// TwinCAT 3 PLC project SFICrane
// ProgramVersion: 3.1.4023.0
// libraries:
//   Tc2_MC2, * (Beckhoff Automation GmbH)
//   Tc2_MC2_Drive, * (Beckhoff Automation GmbH)
//   Tc2_Standard, * (Beckhoff Automation GmbH)
//   Tc2_System, * (Beckhoff Automation GmbH)
//   Tc2_Utilities, * (Beckhoff Automation GmbH)
//   Tc3_Module, * (Beckhoff Automation GmbH)
// project tree:
//   AXIS CONTROL/ GVL_AXIS1.TcGVL, GVL_AXIS2.TcGVL (not stored), GVL_AXIS3.TcGVL, GVL_AXIS4.TcGVL, GVL_Safety_AXIS4.TcGVL, P_AxisControl.TcPOU, P_AxisControl_1.TcPOU, ST_MC_CMD.TcDUT (not stored), ST_MC_ParametersAxis.TcDUT (not stored), ST_MC_Status.TcDUT (not stored)
//   / GlobalTextList.TcGTLO, MAIN.TcPOU (not stored), PlcTask.TcTTO (not stored), Visualization Manager.TcVMO (not stored)
//   HMI/ HMI.TcVIS
//   INPUTS/Function Blocks/ FB_AnalogInputScaling.TcPOU (not stored), FB_JoystickInputScaling.TcPOU (not stored)
//   INPUTS/ G_Inputs.TcGVL, G_ScalingParameters.TcGVL (not stored), G_Sensors.TcGVL (not stored), P_Inputs.TcPOU
//   INPUTS/Struct/ ST_AnalogInput.TcDUT (not stored), ST_AnalogInputScaling.TcDUT (not stored), ST_AnalogInputStatus.TcDUT (not stored), ST_JoystickInputScaling.TcDUT (not stored), ST_Parameters.TcDUT (not stored)
//   MACHINE CONTROL/ G_MachineControl.TcGVL, P_MachineControl.TcPOU (unreadable)
//   MACHINE CONTROL/KinematicFunctions2d/ cosd.TcPOU (not stored), FB_Forward.TcPOU, GVL_InverseKinematics.TcGVL, FB_Inverse.TcPOU (not stored), rt_ceild.TcPOU (not stored), rt_floord.TcPOU (not stored), rt_remd.TcPOU (not stored), FB_WireLengthOnCraneFunction.TcPOU (not stored)
//   OUTPUTS/ G_Outputs.TcGVL, P_Outputs.TcPOU (not stored)
//   StablePlatform/ FB_AnalogInputScalingPlusMinus.TcPOU (not stored), fPlatformAngleTheta1.TcPOU, P_StablePlatform.TcPOU
//   StablePlatform/Function Blocks/ FB_AnalogInputScaling_1.TcPOU (not stored), FB_JoystickInputScaling_1.TcPOU, FB_ValveOutput.TcPOU
//   StablePlatform/GVL/ G_StablePlatformIO.TcGVL, G_StablePlatformParameters.TcGVL, G_StablePlatformScaledIO.TcGVL
//   StablePlatform/Struct/ ST_AnalogInputScaling_1.TcDUT, ST_JoystickInputScaling_1.TcDUT, ST_ValveDeadBand.TcDUT, ST_ValveOutput.TcDUT

// ---- StablePlatform/Struct/ST_AnalogInputScaling_1.TcDUT
TYPE ST_AnalogInputScaling_1 :
STRUCT
	fMaxInputValue 			: LREAL;	// tunable max input value 
	fMinInputValue			: LREAL;	// tunable min input value  
	fMaxOutputValue  		: LREAL;	// max sensor output value
	fMinOutputValue  		: LREAL;	// min sensor output value	
END_STRUCT
END_TYPE

// ---- StablePlatform/Struct/ST_JoystickInputScaling_1.TcDUT
TYPE ST_JoystickInputScaling_1 :
STRUCT
	fMaxInputValue			: LREAL;	// tunable max input value
	fMinInputValue 			: LREAL;	// tunable min input value
	fNeutralInputValue  	: LREAL;	// tunable neutral input value
	fNeutralDeadband		: LREAL;	// tunable dead_band value
	fMaxOutputValue  		: LREAL;	// normalized max output value
	fMinOutputValue  		: LREAL;	// normalized min output value
	fNeutralOutputValue  	: LREAL;	// normalized neutral output value
END_STRUCT
END_TYPE

// ---- StablePlatform/Struct/ST_ValveDeadBand.TcDUT
TYPE ST_ValveDeadBand :
STRUCT
	fPosMax	: LREAL; // Positive min value [19660..29490]
	fPosMin	: LREAL; // Positive max value [19660..29490]
	fNegMin : LREAL; // Negative max value [9830..19660]
	fNegMax	: LREAL; // Negative min value [9830..19660]
END_STRUCT
END_TYPE

// ---- StablePlatform/Struct/ST_ValveOutput.TcDUT
TYPE ST_ValveOutput :
STRUCT
	bEnable					AT %Q* : BOOL := 0;
	nValveOutput 			AT %Q* : INT := 19660;
END_STRUCT
END_TYPE

// ---- AXIS CONTROL/GVL_AXIS1.TcGVL
{attribute 'qualified_only'}
VAR_GLOBAL

//Axis1 Bottom Cylinder 'BC'
BCAxis : AXIS_REF;

//Motion Control Function Block Instant Variable 
fbBC_Reset				: MC_Reset;
fbBC_Power				: MC_Power;
fbBC_Home				: MC_Home;
fbBC_Jog				: MC_Jog;
fbBC_MoveVelocity		: MC_MoveVelocity;
fbBC_Stop				: MC_Stop;
fbBC_MoveAbs			: MC_MoveAbsolute;
fbBC_ExtSetDis			: MC_ExtSetPointGenDisable;
fbBC_ExtSetEnab			: MC_ExtSetPointGenEnable;
fbBC_Rtrig				: R_TRIG;
fbBC_SetReset			: SR;
fbBC_ResetSet			: RS;


//Input: Command
bBC_ResetExe			: BOOL;

bBC_PowerEnCmd			: BOOL;
bBC_PowerEnPositive		: BOOL;
bBC_PowerEnNegative 	: BOOL;

bBC_HomeExe				: BOOL;
bBC_HomeCamInput		: BOOL;

bBC_JogFwd				: BOOL;
bBC_JogRev				: BOOL;	

bBC_MoveVelExe			: BOOL;
	
bBC_StopExe				: BOOL;

bBC_MoveAbsExe			: BOOL;

bBC_MoveContAbsExe		: BOOL;

bBC_MoveContAbsInEndVel	: BOOL;

bBC_MoveAddExe			: BOOL;

bBC_ExtSetGenDisExe		: BOOL;
bBC_ExtSetGenEnaExe		: BOOL;

bBC_MoveAbsDone			: BOOL;

fBC_ExtSetFeedDirection	: DINT;

fBC_MoveContAbsExeTrig	: UINT;


stBC_VelCmd				: ST_MC_CMD := (bExe := FALSE, lrVelocity := 100);//, EnuDirection := MC_Positive_Direction); 
//stBC_VelCmd				: ST_MC_CMD := (bExe := FALSE, lrVelocity := 100, lrAcceleration := 0, lrDeceleration := 0, lrJerk := 0, lrDistance := 0, lrPosition := 0, EnuDirection := MC_Positive_Direction, EnuBufferMode := 0, EnuOptions := 0 ); 

//Variables/Parameters
lrBC_PowerOverride		: LREAL;
lrBC_HomePosition		: LREAL;
lrBC_JogVelocity		: LREAL;
lrBC_MoveVelVelocity	: LREAL;
lrBC_MoveAbsPosition	: LREAL;
lrBC_MoveAbsVelocity	: LREAL;
lrBC_MoveContAbsPos		: LREAL;
lrBC_MoveContAbsEndVel 	: LREAL := 0;
lrBC_MoveAddPos			: LREAL;
lrBC_ActPos					AT %I* : LREAL;
lrBC_PosError			: LREAL;
lrBC_VelContrGain		: LREAL := 1.0;
lrBC_ControllerVelRef	: LREAL;

//Direction
//EnuMoveVelDirection		: MC_Direction;

// Status
stBC_Reset				: ST_MC_Status;
stBC_Power				: ST_MC_Status;
stBC_Home				: ST_MC_Status;
stBC_Jog				: ST_MC_Status;
stBC_MoveVelocity		: ST_MC_Status;
stBC_Stop				: ST_MC_Status;
stBC_MoveAbs			: ST_MC_Status;
stBC_MoveContAbs		: ST_MC_Status;
stBC_MoveAdd			: ST_MC_Status;
stBC_ExtSetDis			: ST_MC_Status;
stBC_ExtSetEnab			: ST_MC_Status;
stBC_ExtSetFeed			: ST_MC_Status;

END_VAR

// ---- AXIS CONTROL/GVL_AXIS3.TcGVL
{attribute 'qualified_only'}
VAR_GLOBAL

//Axis3 Top Cylinder 'TC'
TCAxis : AXIS_REF;

//Motion Control Function Block Instant Variable 
fbTC_Reset				: MC_Reset;
fbTC_Power				: MC_Power;
fbTC_Home				: MC_Home;
fbTC_Jog				: MC_Jog;
fbTC_MoveVelocity		: MC_MoveVelocity;
fbTC_Stop				: MC_Stop;
fbTC_MoveAbs			: MC_MoveAbsolute;
fbTC_ExtSetDis			: MC_ExtSetPointGenDisable;
fbTC_ExtSetEnab			: MC_ExtSetPointGenEnable;
fbTC_Rtrig				: R_TRIG;
fbTC_SetReset			: SR;
fbTC_ResetSet			: RS;

//Input: Command
bTC_ResetExe			: BOOL;

bTC_PowerEnCmd			: BOOL;
bTC_PowerEnPositive		: BOOL;
bTC_PowerEnNegative 	: BOOL;

bTC_HomeExe				: BOOL;
bTC_HomeCamInput		: BOOL;

bTC_JogFwd				: BOOL;
bTC_JogRev				: BOOL;	

bTC_MoveVelExe			: BOOL;
	
bTC_StopExe				: BOOL;

bTC_MoveAbsExe			: BOOL;

bTC_ExtSetGenDisExe		: BOOL;
bTC_ExtSetGenEnaExe		: BOOL;

bTC_MoveAbsDone			: BOOL;

fTC_ExtSetFeedDirection	: DINT;

fTC_MoveContAbsExeTrig	: UINT;

stTC_VelCmd				: ST_MC_CMD := (bExe := FALSE, lrVelocity := 100, EnuDirection := MC_Positive_Direction); 
//stTC_VelCmd				: ST_MC_CMD := (bExe := FALSE, lrVelocity := 100, lrAcceleration := 0, lrDeceleration := 0, lrJerk := 0, lrDistance := 0, lrPosition := 0, EnuDirection := MC_Positive_Direction, EnuBufferMode := 0, EnuOptions := 0 ); 

//Variables/Parameters
lrTC_PowerOverride		: LREAL;
lrTC_HomePosition		: LREAL;
lrTC_SetPosition		: LREAL;
lrTC_JogVelocity		: LREAL;
lrTC_MoveVelVelocity	: LREAL;
lrTC_MoveAbsPosition	: LREAL;
lrTC_MoveAbsVelocity	: LREAL;
lrTC_MoveAddPos			: LREAL;

//Direction
EnuMoveVelDirection		: MC_Direction;

// Status
stTC_Reset				: ST_MC_Status;
stTC_Power				: ST_MC_Status;
stTC_Home				: ST_MC_Status;
stTC_SetPosition		: ST_MC_Status;
stTC_Jog				: ST_MC_Status;
stTC_MoveVelocity		: ST_MC_Status;
stTC_Stop				: ST_MC_Status;
stTC_MoveAbs			: ST_MC_Status;
stTC_ExtSetDis			: ST_MC_Status;
stTC_ExtSetEnab			: ST_MC_Status;
stTC_ExtSetFeed			: ST_MC_Status;

END_VAR

// ---- AXIS CONTROL/GVL_AXIS4.TcGVL
{attribute 'qualified_only'}
VAR_GLOBAL

//Axis4 Winch Motor 'WM'
WMAxis : AXIS_REF;

//Motion Control Function Block Instant Variable 
fbWM_Reset				: MC_Reset;
fbWM_Power				: MC_Power;
fbWM_Home				: MC_Home;
fbWM_Jog				: MC_Jog;
fbWM_MoveVelocity		: MC_MoveVelocity;
fbWM_Stop				: MC_Stop;
fbWM_MoveAbs			: MC_MoveAbsolute;

//Input: Command
bWM_ResetExe			: BOOL;

bWM_PowerEnCmd			: BOOL;
bWM_PowerEnPositive		: BOOL;
bWM_PowerEnNegative 	: BOOL;

bWM_HomeExe				: BOOL;
bWM_HomeCamInput		: BOOL;

bWM_JogFwd				: BOOL;
bWM_JogRev				: BOOL;	

bWM_MoveVelExe			: BOOL;
	
bWM_StopExe				: BOOL;

bWM_MoveAbsExe			: BOOL;

stWM_VelCmd				: ST_MC_CMD := (bExe := FALSE, lrVelocity := 100, EnuDirection := MC_Positive_Direction); 
//stWM_VelCmd				: ST_MC_CMD := (bExe := FALSE, lrVelocity := 100, lrAcceleration := 0, lrDeceleration := 0, lrJerk := 0, lrDistance := 0, lrPosition := 0, EnuDirection := MC_Positive_Direction, EnuBufferMode := 0, EnuOptions := 0 ); 

//Variables/Parameters
lrWM_PowerOverride		: LREAL;
lrWM_HomePosition		: LREAL;
lrWM_SetPosition		: LREAL;
lrWM_JogVelocity		: LREAL;
lrWM_MoveVelVelocity	: LREAL;
lrWM_MoveAbsPosition	: LREAL;

//Direction
EnuMoveVelDirection		: MC_Direction;

// Status
stWM_Reset				: ST_MC_Status;
stWM_Power				: ST_MC_Status;
stWM_Home				: ST_MC_Status;
stWM_SetPosition		: ST_MC_Status;
stWM_Jog				: ST_MC_Status;
stWM_MoveVelocity		: ST_MC_Status;
stWM_Stop				: ST_MC_Status;
stWM_MoveAbs			: ST_MC_Status;

//Safety
bInAckSignal		AT %I*	:BOOL;


END_VAR

// ---- AXIS CONTROL/GVL_Safety_AXIS4.TcGVL
{attribute 'qualified_only'}
VAR_GLOBAL
	
	bWinchMotor24vDisable AT %Q* : BOOL;
	TwinSafeGroupComErrAck AT %Q* : BOOL; 
	TwinSafeGroupRunStop AT %Q* : BOOL := TRUE; 
	ChA_STO_Enable AT %Q* : BOOL;
	ChA_STO_Active AT %I* : BOOL;  
END_VAR

// ---- INPUTS/G_Inputs.TcGVL
{attribute 'qualified_only'}
VAR_GLOBAL
	bManualModeSelector			AT %I* : BOOL;
	bAutoModeSelector			AT %I* : BOOL;
	bRedButton					AT %I* : BOOL;
	bGreenButton				AT %I* : BOOL;
	bJoystickLeftEnable			AT %I* : BOOL;
	bJoystickRightEnable		AT %I* : BOOL;
	bSafetyRelayRestartButton   AT %I* : BOOL;
	
	// Analog Inputs
	stJoyLX 					: ST_AnalogInput;
	stJoyLY						: ST_AnalogInput;
	stJoyRX 					: ST_AnalogInput;
	stJoyRY						: ST_AnalogInput;

END_VAR

// ---- MACHINE CONTROL/G_MachineControl.TcGVL
{attribute 'qualified_only'}
VAR_GLOBAL
	bManualMode 			: BOOL;
	bAutoMode 				: BOOL;
	bWinchEnable 			: BOOL;
	bCylEnable 				: BOOL;
	fWinchControlInput 		: LREAL;
	fWinchTime				: LREAL;
	fCylControlInput 		: LREAL;
	fCylTime				: LREAL;
	fVelRefWinch 			: LREAL;
	fPosRefWinch 			: LREAL;
	fControlSignWinch		: LREAL;
	fVelRefCyl 				: LREAL;
	fPosRefCyl 				: LREAL;
	fControlSignCyl			: LREAL;
	fPositionErrorWinch_mm 	: LREAL;
	fPositionErrorCylinder_mm : LREAL;
	fSampleTime				: LREAL := 0.002;
	fTimeSinceStart			: LREAL := 0.0;
	fStrokeActuatorMain 	AT %I* : LREAL;
	fStrokeActuatorKnuckle 	AT %I* : LREAL;
	fSlewMotorAngle			AT %I* : LREAL;
	fWinchMotorAngle		AT %I* : LREAL;	
<<<<<<< HEAD:TwinCAT/SFICraneNewSetup/SFICrane/MACHINE CONTROL/G_Work.TcGVL
	bEMG_Restart 			AT %Q* : BOOL;
=======
	fWinchAngle				: LREAL;
	
	fCraneForwardY 			: LREAL;
	fTheta3Forward			: LREAL;
	fTheta4Forward			: LREAL;
	fWireLengthOnCrane		: LREAL;
	fEncoderValue0Turns		: LREAL;
	fEncoderValue5Turns		: LREAL;
	fEncoderValueLayer2		: LREAL;
	fEncoderValuePayload0	: LREAL;
	fPayloadHeightIni		: LREAL := 1.0;
	fWinchPitchRadiusLayer1 : LREAL := 0.0716;
	fWinchPitchRadiusLayer2 : LREAL := 0.0731;
	fWinchGearRatio 		: LREAL := 32;
	fWinchMotorAngleRef			: LREAL;
>>>>>>> edf6f2e068e7575cdf7fdcbf34452a62e6a1fd5d:TwinCAT/SFICraneNewSetup/SFICrane/MACHINE CONTROL/G_MachineControl.TcGVL
END_VAR

// ---- MACHINE CONTROL/KinematicFunctions2d/GVL_InverseKinematics.TcGVL
{attribute 'qualified_only'}
VAR_GLOBAL
	fTooltipXCoordGlobalIni: LREAL := 2.8;
	fTooltipYCoordGlobalIni: LREAL := 2.2;
	
	fTheta1 : LREAL := 0;
	fAngleMainArmInverse :	LREAL;
	fAngleKnuckleArmInverse : LREAL;
	fStrokeActuatorMainInverse : LREAL;
	fStrokeActuatorKnuckleInverse : LREAL;
END_VAR

// ---- OUTPUTS/G_Outputs.TcGVL
{attribute 'qualified_only'}
VAR_GLOBAL
	// PLC Rack
	
	// RIO Rack
	// Digital Outputs
	bGreenButtonLight 			AT %Q* : BOOL;
	bRedButtonLight 			AT %Q* : BOOL;
	// Analog Outputs
	//stWinchValveOutput 		: ST_ValveOutput;
	//stCylValveOutput 			: ST_ValveOutput;
END_VAR

// ---- StablePlatform/GVL/G_StablePlatformIO.TcGVL
{attribute 'qualified_only'}
VAR_GLOBAL
	bSVEnable AT %Q* : BOOL; 
	nSVControlSignal AT %Q* : INT; 
	//fJoyLeftX AT %I* : INT; 
	
	//bJoyLeftPushButton AT %I* : BOOL; 
	
	npA AT %I* : INT;
	npB AT %I* : INT;
	npS AT %I* : INT;
	
	nSVFeedback AT %I* : INT;
	
	bModeSwitchOff AT %I* : BOOL;
	
	nPistonPosition AT %I* : INT;
	nPistonVelocity AT %I* : INT;
END_VAR

// ---- StablePlatform/GVL/G_StablePlatformParameters.TcGVL
{attribute 'qualified_only'}
VAR_GLOBAL
	stPressureSensorScaling400bar 	: ST_AnalogInputScaling := (fMaxInputValue := 32767.0, fMinInputValue := 0.0, fMaxOutputValue := 400.0, fMinOutputValue := 0.0);
	stJoystickInputScalingX 		: ST_JoystickInputScaling := (fMaxInputValue := 20625.0, fMinInputValue := 11800.0, fNeutralInputValue := 16265, fNeutralDeadband := 100.0, fMaxOutputValue := 1.0, fMinOutputValue := -1.0, fNeutralOutputValue := 0.0);
	stSVValveDeadBand 				: ST_ValveDeadBand := (fPosMax := 29490.0, fPosMin := 20950.0, fNegMin := 18250.0, fNegMax := 9830.0);
	stSVFeedbackScaling 			: ST_AnalogInputScaling := (fMaxInputValue := 32767.0, fMinInputValue := 0.0, fMaxOutputValue := 20.0, fMinOutputValue := 4.0);
END_VAR

// ---- StablePlatform/GVL/G_StablePlatformScaledIO.TcGVL
{attribute 'qualified_only'}
VAR_GLOBAL
	bpA : LREAL; // 0..400bar
	bpB : LREAL; // 0..400bar
	bpS : LREAL; // 0..400bar
	fSVFeedback : LREAL; // 4..20 mA  | 0 = fault/off
	fJoystickNormalizedX : LREAL; // -1..0..1
END_VAR

// ---- AXIS CONTROL/P_AxisControl.TcPOU
PROGRAM P_AxisControl
VAR
END_VAR

//Axis Control program based on youtube series Twincat 3 NC Videos MB05a until MB17b plus MB22 by @electricalautomation https://www.youtube.com/watch?v=BxRAOdTks9I&list=PL762SfoJC-e8NbAUQ-H7a_TOdqrlBPCw4&index=25

IF G_Inputs.bManualModeSelector THEN
	Manual_mode();
ELSIF G_Inputs.bAutoModeSelector THEN
	Auto_mode();
ELSE
	GVL_AXIS1.lrBC_PowerOverride := 0;
	GVL_AXIS1.bBC_StopExe := TRUE;
	GVL_AXIS2.lrSJ_PowerOverride := 0;
	GVL_AXIS2.bSJ_StopExe := TRUE;
	GVL_AXIS3.lrTC_PowerOverride := 0;
	GVL_AXIS3.bTC_StopExe := TRUE;
	GVL_AXIS4.lrWM_PowerOverride := 0;
	GVL_AXIS4.bWM_StopExe := TRUE;
END_IF

METHOD Auto_mode : BOOL
VAR_INPUT
END_VAR
//AXIS 1 Main arm actuator

GVL_AXIS1.lrBC_PowerOverride := 100;

GVL_AXIS1.bBC_ResetExe := G_Inputs.bJoystickLeftEnable OR G_Inputs.bGreenButton OR GVL_AXIS1.bBC_MoveAbsDone;

//Power Enable
GVL_AXIS1.bBC_PowerEnCmd := G_Inputs.bAutoModeSelector;
GVL_AXIS1.bBC_PowerEnNegative := G_Inputs.bAutoModeSelector;
GVL_AXIS1.bBC_PowerEnPositive := G_Inputs.bAutoModeSelector;

GVL_AXIS1.lrBC_MoveAbsPosition := GVL_InverseKinematics.fStrokeActuatorMainInverse*1000;
GVL_AXIS1.lrBC_MoveAbsVelocity := 30;
GVL_AXIS1.bBC_MoveAbsExe := G_Inputs.bGreenButton;


//Position control
IF G_Inputs.bJoystickLeftEnable AND GVL_AXIS1.bBC_MoveAbsDone THEN
	GVL_AXIS1.bBC_ExtSetGenDisExe := FALSE;
	GVL_AXIS1.bBC_ExtSetGenEnaExe := TRUE;
ELSE
	GVL_AXIS1.bBC_ExtSetGenDisExe := TRUE;
	GVL_AXIS1.bBC_ExtSetGenEnaExe := FALSE;
END_IF


GVL_AXIS1.lrBC_MoveAddPos := GVL_InverseKinematics.fStrokeActuatorMainInverse*1000;


//Update axis
AXIS1_LD_Auto();


//Axis 3 Knuckle arm actuator

GVL_AXIS3.lrTC_PowerOverride := 100;

GVL_AXIS3.bTC_ResetExe := G_Inputs.bJoystickLeftEnable OR G_Inputs.bGreenButton OR GVL_AXIS3.bTC_MoveAbsDone;

//Power Enable
GVL_AXIS3.bTC_PowerEnCmd := G_Inputs.bAutoModeSelector;
GVL_AXIS3.bTC_PowerEnNegative := G_Inputs.bAutoModeSelector;
GVL_AXIS3.bTC_PowerEnPositive := G_Inputs.bAutoModeSelector;

GVL_AXIS3.lrTC_MoveAbsPosition := GVL_InverseKinematics.fStrokeActuatorKnuckleInverse*1000;
GVL_AXIS3.lrTC_MoveAbsVelocity := 30;
GVL_AXIS3.bTC_MoveAbsExe := G_Inputs.bGreenButton;


//Position control
IF G_Inputs.bJoystickLeftEnable AND GVL_AXIS3.bTC_MoveAbsDone THEN
	GVL_AXIS3.bTC_ExtSetGenDisExe := FALSE;
	GVL_AXIS3.bTC_ExtSetGenEnaExe := TRUE;
ELSE
	GVL_AXIS3.bTC_ExtSetGenDisExe := TRUE;
	GVL_AXIS3.bTC_ExtSetGenEnaExe := FALSE;
END_IF


GVL_AXIS3.lrTC_MoveAddPos := GVL_InverseKinematics.fStrokeActuatorKnuckleInverse*1000;


//Update axis
AXIS3_LD_Auto();


//Axis 4 Winch motor

GVL_AXIS4.lrWM_PowerOverride := 100;

GVL_AXIS4.bWM_ResetExe := G_Inputs.bJoystickRightEnable OR G_Inputs.bGreenButton OR GVL_AXIS1.bBC_MoveAbsDone;

//Power Enable
GVL_AXIS4.bWM_PowerEnCmd := G_Inputs.bAutoModeSelector;
GVL_AXIS4.bWM_PowerEnNegative := G_Inputs.bAutoModeSelector;
GVL_AXIS4.bWM_PowerEnPositive := G_Inputs.bAutoModeSelector;


GVL_AXIS4.lrWM_MoveAbsPosition := G_MachineControl.fWinchMotorAngleRef;
GVL_AXIS4.lrWM_MoveAbsVelocity := 10;
GVL_AXIS4.bWM_MoveAbsExe := G_Inputs.bGreenButton;


//Position control
IF G_Inputs.bJoystickRightEnable AND GVL_AXIS4.bWM_MoveAbsDone  THEN
	GVL_AXIS4.bWM_ExtSetGenDisExe := FALSE;
	GVL_AXIS4.bWM_ExtSetGenEnaExe := TRUE;
ELSE
	GVL_AXIS4.bWM_ExtSetGenDisExe := TRUE;
	GVL_AXIS4.bWM_ExtSetGenEnaExe := FALSE;
END_IF

(*
//Position control
IF G_Inputs.bJoystickRightEnable THEN
	GVL_AXIS4.bWM_ExtSetGenDisExe := FALSE;
	GVL_AXIS4.bWM_ExtSetGenEnaExe := TRUE;
ELSE
	GVL_AXIS4.bWM_ExtSetGenDisExe := TRUE;
	GVL_AXIS4.bWM_ExtSetGenEnaExe := FALSE;
END_IF
*)

GVL_AXIS4.lrWM_MoveAddPos := G_MachineControl.fPosRefWinch*180/PI; //Convert to degrees


//Update axis
AXIS4_LD_Auto();
END_METHOD

METHOD AXIS1_LD : BOOL
VAR_INPUT
END_VAR
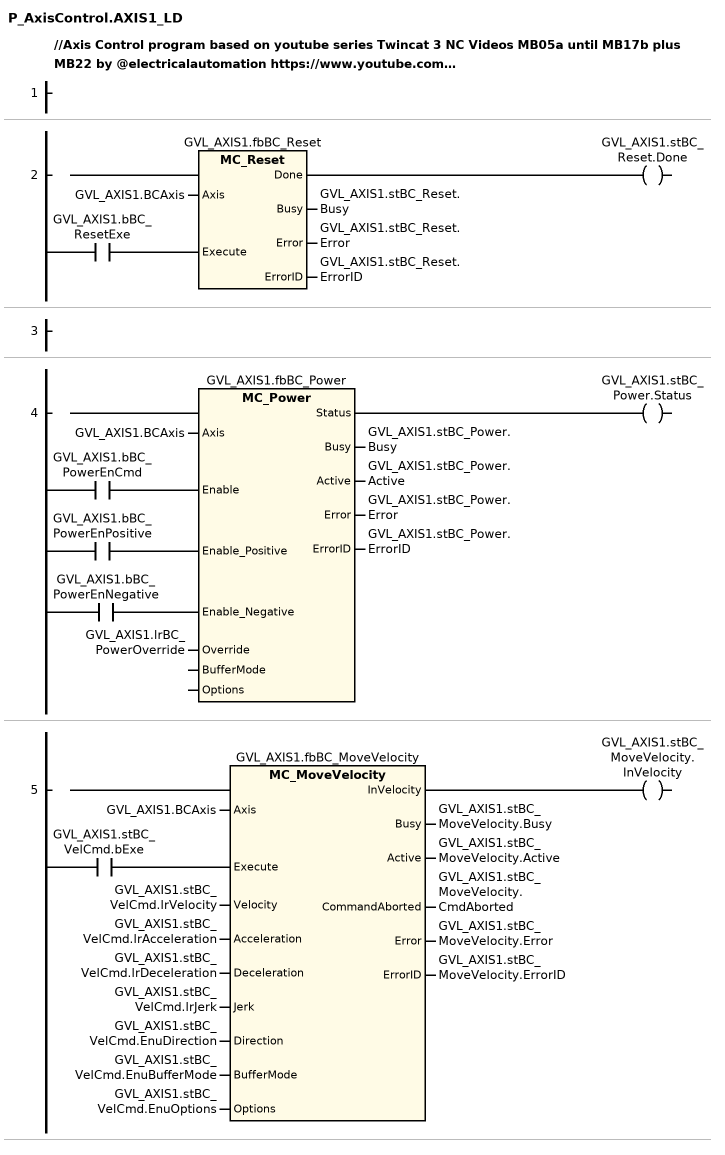
// NETWORK 1: //Axis Control program based on youtube series Twincat 3 NC Videos MB05a until MB17b plus MB22 by @electricalautomation https://www.youtube.com/watch?v=BxRAOdTks9I&list=PL762SfoJC-e8NbAUQ-H7a_TOdqrlBPCw4&index=25

// NETWORK 2
GVL_AXIS1.fbBC_Reset(
    Axis := GVL_AXIS1.BCAxis,
    Execute := GVL_AXIS1.bBC_ResetExe,
    Busy => GVL_AXIS1.stBC_Reset.Busy,
    Error => GVL_AXIS1.stBC_Reset.Error,
    ErrorID => GVL_AXIS1.stBC_Reset.ErrorID); // MC_Reset
GVL_AXIS1.stBC_Reset.Done := GVL_AXIS1.fbBC_Reset.Done;

// NETWORK 3

// NETWORK 4
GVL_AXIS1.fbBC_Power(
    Axis := GVL_AXIS1.BCAxis,
    Enable := GVL_AXIS1.bBC_PowerEnCmd,
    Enable_Positive := GVL_AXIS1.bBC_PowerEnPositive,
    Enable_Negative := GVL_AXIS1.bBC_PowerEnNegative,
    Override := GVL_AXIS1.lrBC_PowerOverride,
    Busy => GVL_AXIS1.stBC_Power.Busy,
    Active => GVL_AXIS1.stBC_Power.Active,
    Error => GVL_AXIS1.stBC_Power.Error,
    ErrorID => GVL_AXIS1.stBC_Power.ErrorID); // MC_Power
GVL_AXIS1.stBC_Power.Status := GVL_AXIS1.fbBC_Power.Status;

// NETWORK 5
GVL_AXIS1.fbBC_MoveVelocity(
    Axis := GVL_AXIS1.BCAxis,
    Execute := GVL_AXIS1.stBC_VelCmd.bExe,
    Velocity := GVL_AXIS1.stBC_VelCmd.lrVelocity,
    Acceleration := GVL_AXIS1.stBC_VelCmd.lrAcceleration,
    Deceleration := GVL_AXIS1.stBC_VelCmd.lrDeceleration,
    Jerk := GVL_AXIS1.stBC_VelCmd.lrJerk,
    Direction := GVL_AXIS1.stBC_VelCmd.EnuDirection,
    BufferMode := GVL_AXIS1.stBC_VelCmd.EnuBufferMode,
    Options := GVL_AXIS1.stBC_VelCmd.EnuOptions,
    Busy => GVL_AXIS1.stBC_MoveVelocity.Busy,
    Active => GVL_AXIS1.stBC_MoveVelocity.Active,
    CommandAborted => GVL_AXIS1.stBC_MoveVelocity.CmdAborted,
    Error => GVL_AXIS1.stBC_MoveVelocity.Error,
    ErrorID => GVL_AXIS1.stBC_MoveVelocity.ErrorID); // MC_MoveVelocity
GVL_AXIS1.stBC_MoveVelocity.InVelocity := GVL_AXIS1.fbBC_MoveVelocity.InVelocity;
END_METHOD

METHOD AXIS1_LD_Auto : BOOL
VAR_INPUT
END_VAR
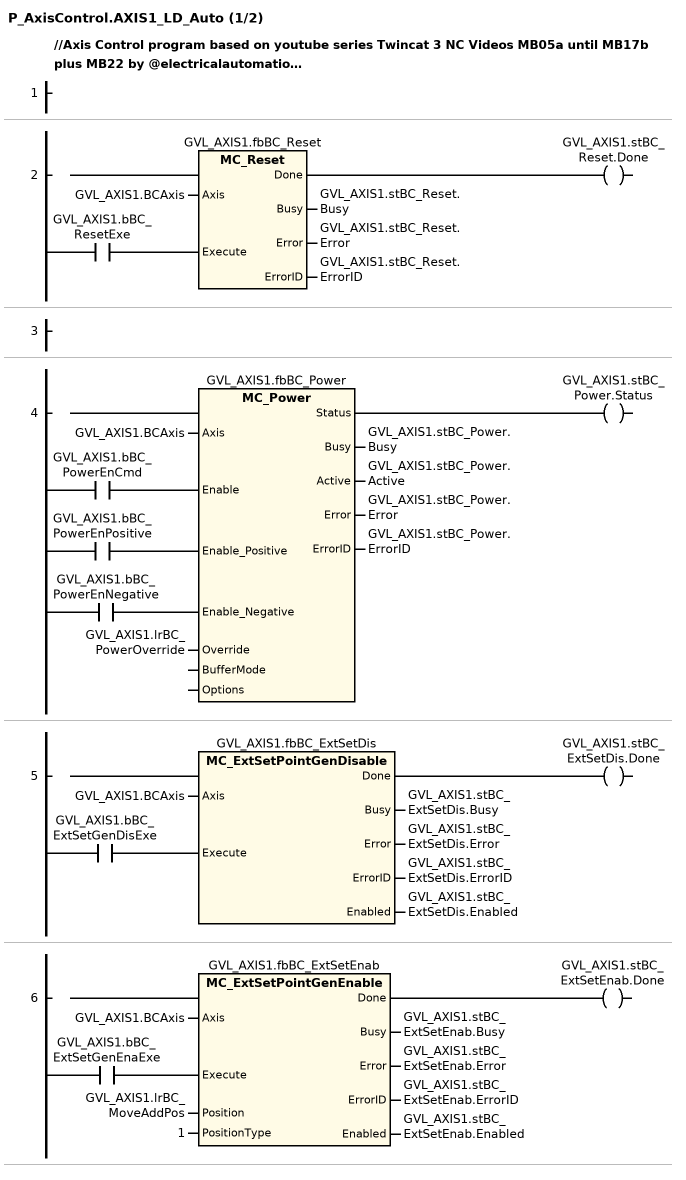
// NETWORK 1: //Axis Control program based on youtube series Twincat 3 NC Videos MB05a until MB17b plus MB22 by @electricalautomation https://www.youtube.com/watch?v=BxRAOdTks9I&list=PL762SfoJC-e8NbAUQ-H7a_TOdqrlBPCw4&index=25

// NETWORK 2
GVL_AXIS1.fbBC_Reset(
    Axis := GVL_AXIS1.BCAxis,
    Execute := GVL_AXIS1.bBC_ResetExe,
    Busy => GVL_AXIS1.stBC_Reset.Busy,
    Error => GVL_AXIS1.stBC_Reset.Error,
    ErrorID => GVL_AXIS1.stBC_Reset.ErrorID); // MC_Reset
GVL_AXIS1.stBC_Reset.Done := GVL_AXIS1.fbBC_Reset.Done;

// NETWORK 3

// NETWORK 4
GVL_AXIS1.fbBC_Power(
    Axis := GVL_AXIS1.BCAxis,
    Enable := GVL_AXIS1.bBC_PowerEnCmd,
    Enable_Positive := GVL_AXIS1.bBC_PowerEnPositive,
    Enable_Negative := GVL_AXIS1.bBC_PowerEnNegative,
    Override := GVL_AXIS1.lrBC_PowerOverride,
    Busy => GVL_AXIS1.stBC_Power.Busy,
    Active => GVL_AXIS1.stBC_Power.Active,
    Error => GVL_AXIS1.stBC_Power.Error,
    ErrorID => GVL_AXIS1.stBC_Power.ErrorID); // MC_Power
GVL_AXIS1.stBC_Power.Status := GVL_AXIS1.fbBC_Power.Status;

// NETWORK 5
GVL_AXIS1.fbBC_ExtSetDis(
    Axis := GVL_AXIS1.BCAxis,
    Execute := GVL_AXIS1.bBC_ExtSetGenDisExe,
    Busy => GVL_AXIS1.stBC_ExtSetDis.Busy,
    Error => GVL_AXIS1.stBC_ExtSetDis.Error,
    ErrorID => GVL_AXIS1.stBC_ExtSetDis.ErrorID,
    Enabled => GVL_AXIS1.stBC_ExtSetDis.Enabled); // MC_ExtSetPointGenDisable
GVL_AXIS1.stBC_ExtSetDis.Done := GVL_AXIS1.fbBC_ExtSetDis.Done;

// NETWORK 6
GVL_AXIS1.fbBC_ExtSetEnab(
    Axis := GVL_AXIS1.BCAxis,
    Execute := GVL_AXIS1.bBC_ExtSetGenEnaExe,
    Position := GVL_AXIS1.lrBC_MoveAddPos,
    PositionType := 1,
    Busy => GVL_AXIS1.stBC_ExtSetEnab.Busy,
    Error => GVL_AXIS1.stBC_ExtSetEnab.Error,
    ErrorID => GVL_AXIS1.stBC_ExtSetEnab.ErrorID,
    Enabled => GVL_AXIS1.stBC_ExtSetEnab.Enabled); // MC_ExtSetPointGenEnable
GVL_AXIS1.stBC_ExtSetEnab.Done := GVL_AXIS1.fbBC_ExtSetEnab.Done;

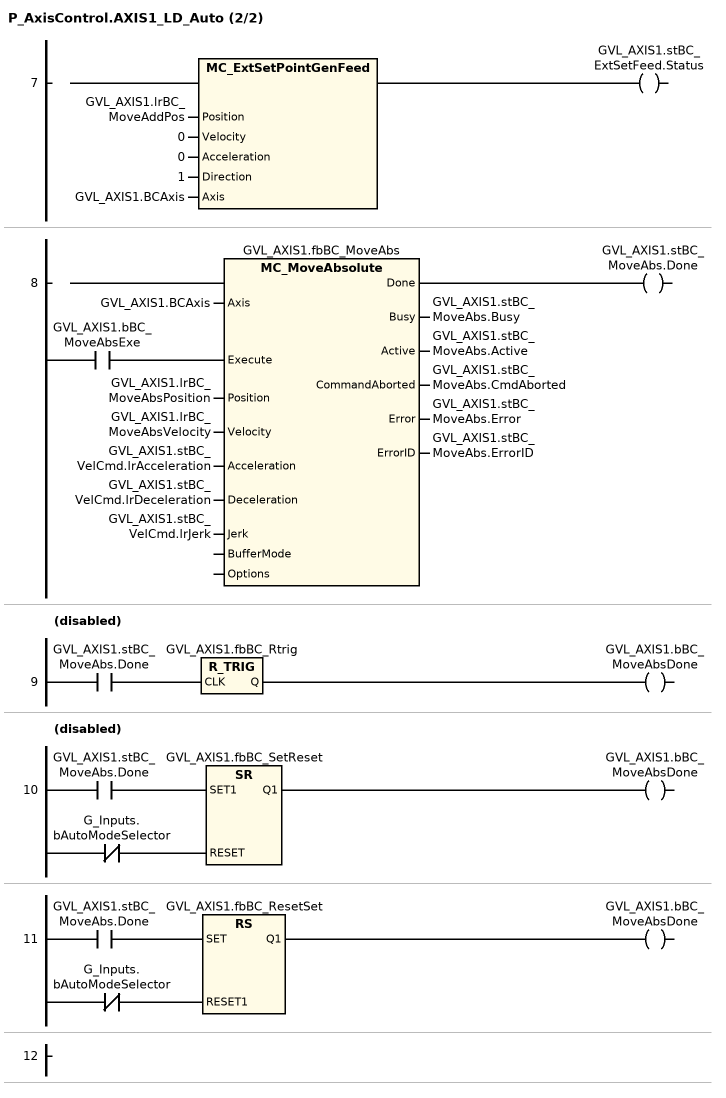
// NETWORK 7
GVL_AXIS1.stBC_ExtSetFeed.Status := MC_ExtSetPointGenFeed(Position := GVL_AXIS1.lrBC_MoveAddPos, Velocity := 0, Acceleration := 0, Direction := 1, Axis := GVL_AXIS1.BCAxis);

// NETWORK 8
GVL_AXIS1.fbBC_MoveAbs(
    Axis := GVL_AXIS1.BCAxis,
    Execute := GVL_AXIS1.bBC_MoveAbsExe,
    Position := GVL_AXIS1.lrBC_MoveAbsPosition,
    Velocity := GVL_AXIS1.lrBC_MoveAbsVelocity,
    Acceleration := GVL_AXIS1.stBC_VelCmd.lrAcceleration,
    Deceleration := GVL_AXIS1.stBC_VelCmd.lrDeceleration,
    Jerk := GVL_AXIS1.stBC_VelCmd.lrJerk,
    Busy => GVL_AXIS1.stBC_MoveAbs.Busy,
    Active => GVL_AXIS1.stBC_MoveAbs.Active,
    CommandAborted => GVL_AXIS1.stBC_MoveAbs.CmdAborted,
    Error => GVL_AXIS1.stBC_MoveAbs.Error,
    ErrorID => GVL_AXIS1.stBC_MoveAbs.ErrorID); // MC_MoveAbsolute
GVL_AXIS1.stBC_MoveAbs.Done := GVL_AXIS1.fbBC_MoveAbs.Done;

// NETWORK 9 (disabled)
// GVL_AXIS1.fbBC_Rtrig(CLK := GVL_AXIS1.stBC_MoveAbs.Done); // R_TRIG
// GVL_AXIS1.bBC_MoveAbsDone := GVL_AXIS1.fbBC_Rtrig.Q;

// NETWORK 10 (disabled)
// GVL_AXIS1.fbBC_SetReset(SET1 := GVL_AXIS1.stBC_MoveAbs.Done, RESET := NOT G_Inputs.bAutoModeSelector); // SR
// GVL_AXIS1.bBC_MoveAbsDone := GVL_AXIS1.fbBC_SetReset.Q1;

// NETWORK 11
GVL_AXIS1.fbBC_ResetSet(SET := GVL_AXIS1.stBC_MoveAbs.Done, RESET1 := NOT G_Inputs.bAutoModeSelector); // RS
GVL_AXIS1.bBC_MoveAbsDone := GVL_AXIS1.fbBC_ResetSet.Q1;

// NETWORK 12
END_METHOD

METHOD AXIS2_LD : BOOL
VAR_INPUT
END_VAR
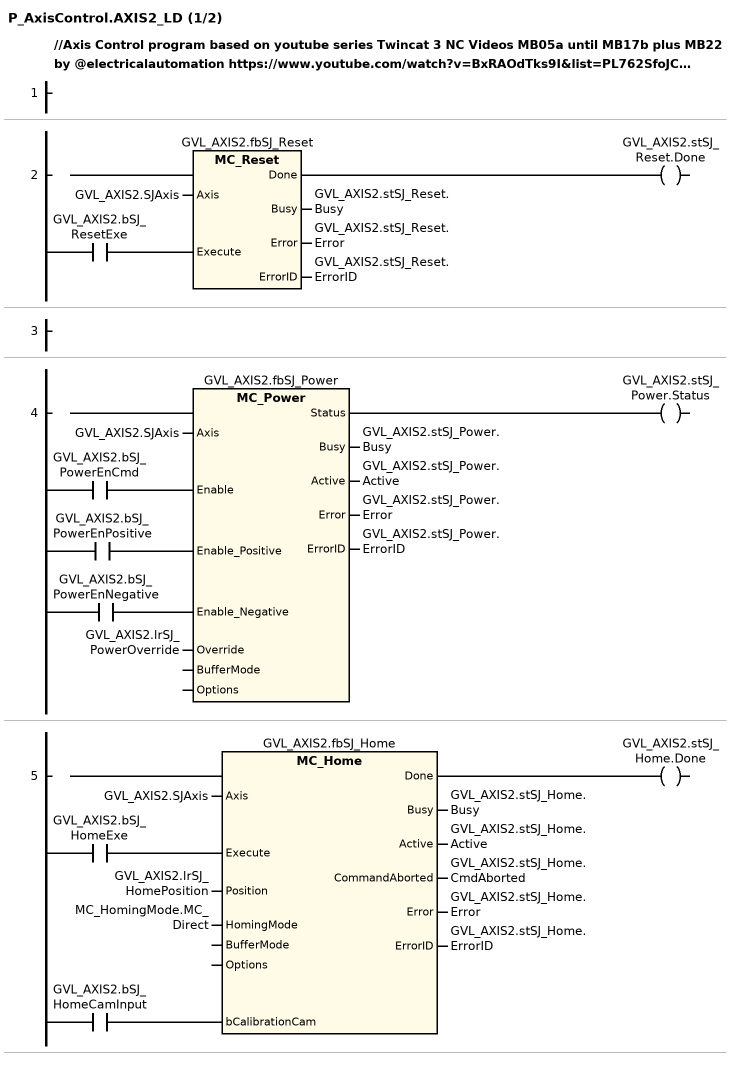
// NETWORK 1: //Axis Control program based on youtube series Twincat 3 NC Videos MB05a until MB17b plus MB22 by @electricalautomation https://www.youtube.com/watch?v=BxRAOdTks9I&list=PL762SfoJC-e8NbAUQ-H7a_TOdqrlBPCw4&index=25

// NETWORK 2
GVL_AXIS2.fbSJ_Reset(
    Axis := GVL_AXIS2.SJAxis,
    Execute := GVL_AXIS2.bSJ_ResetExe,
    Busy => GVL_AXIS2.stSJ_Reset.Busy,
    Error => GVL_AXIS2.stSJ_Reset.Error,
    ErrorID => GVL_AXIS2.stSJ_Reset.ErrorID); // MC_Reset
GVL_AXIS2.stSJ_Reset.Done := GVL_AXIS2.fbSJ_Reset.Done;

// NETWORK 3

// NETWORK 4
GVL_AXIS2.fbSJ_Power(
    Axis := GVL_AXIS2.SJAxis,
    Enable := GVL_AXIS2.bSJ_PowerEnCmd,
    Enable_Positive := GVL_AXIS2.bSJ_PowerEnPositive,
    Enable_Negative := GVL_AXIS2.bSJ_PowerEnNegative,
    Override := GVL_AXIS2.lrSJ_PowerOverride,
    Busy => GVL_AXIS2.stSJ_Power.Busy,
    Active => GVL_AXIS2.stSJ_Power.Active,
    Error => GVL_AXIS2.stSJ_Power.Error,
    ErrorID => GVL_AXIS2.stSJ_Power.ErrorID); // MC_Power
GVL_AXIS2.stSJ_Power.Status := GVL_AXIS2.fbSJ_Power.Status;

// NETWORK 5
GVL_AXIS2.fbSJ_Home(
    Axis := GVL_AXIS2.SJAxis,
    Execute := GVL_AXIS2.bSJ_HomeExe,
    Position := GVL_AXIS2.lrSJ_HomePosition,
    HomingMode := MC_HomingMode.MC_Direct,
    bCalibrationCam := GVL_AXIS2.bSJ_HomeCamInput,
    Busy => GVL_AXIS2.stSJ_Home.Busy,
    Active => GVL_AXIS2.stSJ_Home.Active,
    CommandAborted => GVL_AXIS2.stSJ_Home.CmdAborted,
    Error => GVL_AXIS2.stSJ_Home.Error,
    ErrorID => GVL_AXIS2.stSJ_Home.ErrorID); // MC_Home
GVL_AXIS2.stSJ_Home.Done := GVL_AXIS2.fbSJ_Home.Done;

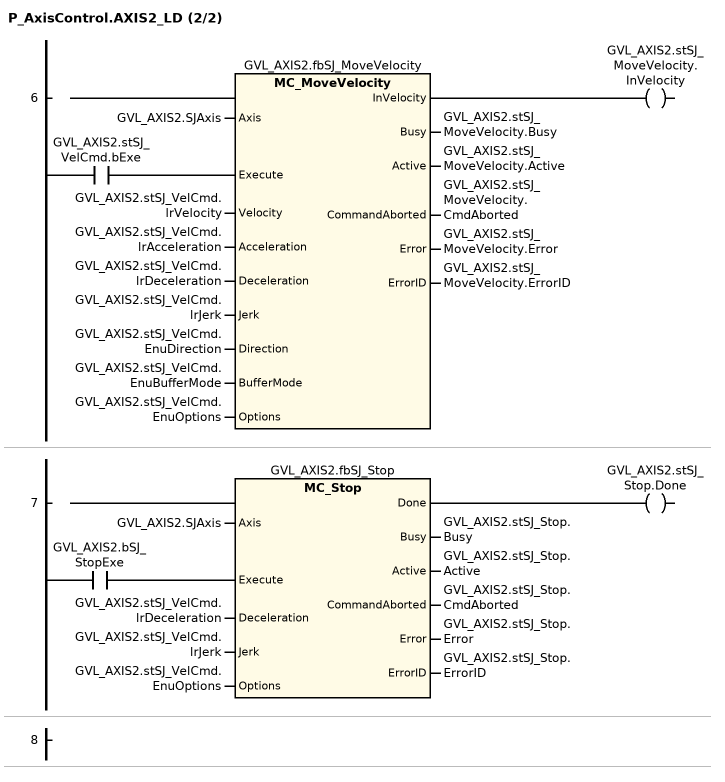
// NETWORK 6
GVL_AXIS2.fbSJ_MoveVelocity(
    Axis := GVL_AXIS2.SJAxis,
    Execute := GVL_AXIS2.stSJ_VelCmd.bExe,
    Velocity := GVL_AXIS2.stSJ_VelCmd.lrVelocity,
    Acceleration := GVL_AXIS2.stSJ_VelCmd.lrAcceleration,
    Deceleration := GVL_AXIS2.stSJ_VelCmd.lrDeceleration,
    Jerk := GVL_AXIS2.stSJ_VelCmd.lrJerk,
    Direction := GVL_AXIS2.stSJ_VelCmd.EnuDirection,
    BufferMode := GVL_AXIS2.stSJ_VelCmd.EnuBufferMode,
    Options := GVL_AXIS2.stSJ_VelCmd.EnuOptions,
    Busy => GVL_AXIS2.stSJ_MoveVelocity.Busy,
    Active => GVL_AXIS2.stSJ_MoveVelocity.Active,
    CommandAborted => GVL_AXIS2.stSJ_MoveVelocity.CmdAborted,
    Error => GVL_AXIS2.stSJ_MoveVelocity.Error,
    ErrorID => GVL_AXIS2.stSJ_MoveVelocity.ErrorID); // MC_MoveVelocity
GVL_AXIS2.stSJ_MoveVelocity.InVelocity := GVL_AXIS2.fbSJ_MoveVelocity.InVelocity;

// NETWORK 7
GVL_AXIS2.fbSJ_Stop(
    Axis := GVL_AXIS2.SJAxis,
    Execute := GVL_AXIS2.bSJ_StopExe,
    Deceleration := GVL_AXIS2.stSJ_VelCmd.lrDeceleration,
    Jerk := GVL_AXIS2.stSJ_VelCmd.lrJerk,
    Options := GVL_AXIS2.stSJ_VelCmd.EnuOptions,
    Busy => GVL_AXIS2.stSJ_Stop.Busy,
    Active => GVL_AXIS2.stSJ_Stop.Active,
    CommandAborted => GVL_AXIS2.stSJ_Stop.CmdAborted,
    Error => GVL_AXIS2.stSJ_Stop.Error,
    ErrorID => GVL_AXIS2.stSJ_Stop.ErrorID); // MC_Stop
GVL_AXIS2.stSJ_Stop.Done := GVL_AXIS2.fbSJ_Stop.Done;

// NETWORK 8
END_METHOD

METHOD AXIS3_LD : BOOL
VAR_INPUT
END_VAR
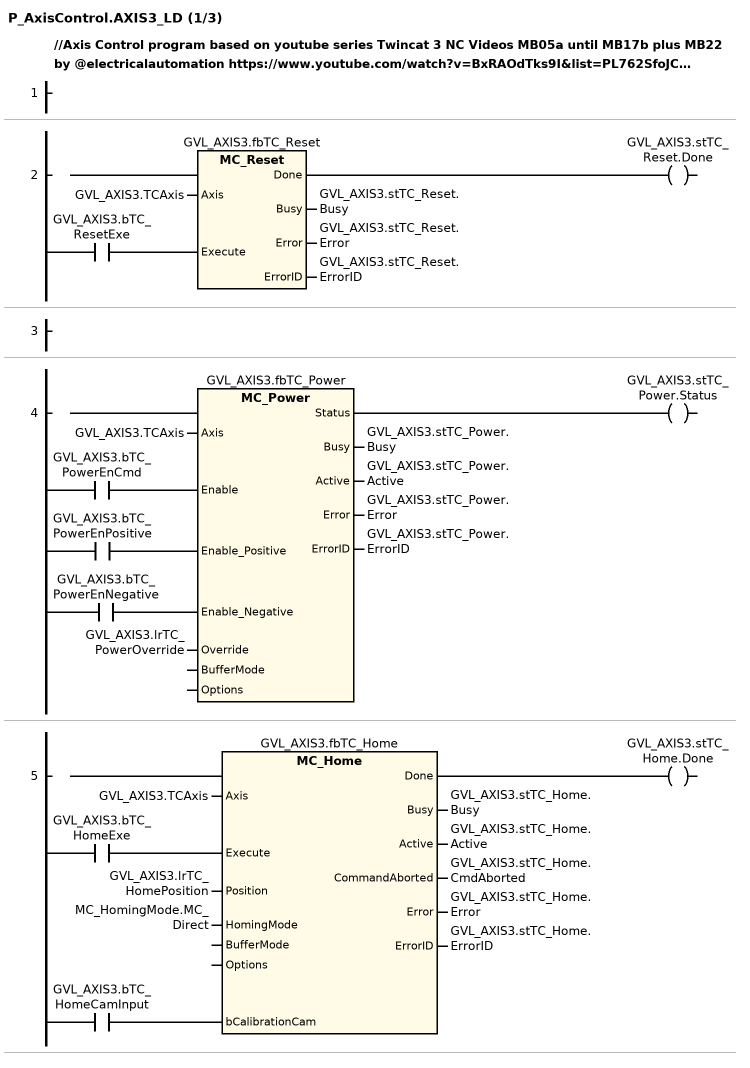
// NETWORK 1: //Axis Control program based on youtube series Twincat 3 NC Videos MB05a until MB17b plus MB22 by @electricalautomation https://www.youtube.com/watch?v=BxRAOdTks9I&list=PL762SfoJC-e8NbAUQ-H7a_TOdqrlBPCw4&index=25

// NETWORK 2
GVL_AXIS3.fbTC_Reset(
    Axis := GVL_AXIS3.TCAxis,
    Execute := GVL_AXIS3.bTC_ResetExe,
    Busy => GVL_AXIS3.stTC_Reset.Busy,
    Error => GVL_AXIS3.stTC_Reset.Error,
    ErrorID => GVL_AXIS3.stTC_Reset.ErrorID); // MC_Reset
GVL_AXIS3.stTC_Reset.Done := GVL_AXIS3.fbTC_Reset.Done;

// NETWORK 3

// NETWORK 4
GVL_AXIS3.fbTC_Power(
    Axis := GVL_AXIS3.TCAxis,
    Enable := GVL_AXIS3.bTC_PowerEnCmd,
    Enable_Positive := GVL_AXIS3.bTC_PowerEnPositive,
    Enable_Negative := GVL_AXIS3.bTC_PowerEnNegative,
    Override := GVL_AXIS3.lrTC_PowerOverride,
    Busy => GVL_AXIS3.stTC_Power.Busy,
    Active => GVL_AXIS3.stTC_Power.Active,
    Error => GVL_AXIS3.stTC_Power.Error,
    ErrorID => GVL_AXIS3.stTC_Power.ErrorID); // MC_Power
GVL_AXIS3.stTC_Power.Status := GVL_AXIS3.fbTC_Power.Status;

// NETWORK 5
GVL_AXIS3.fbTC_Home(
    Axis := GVL_AXIS3.TCAxis,
    Execute := GVL_AXIS3.bTC_HomeExe,
    Position := GVL_AXIS3.lrTC_HomePosition,
    HomingMode := MC_HomingMode.MC_Direct,
    bCalibrationCam := GVL_AXIS3.bTC_HomeCamInput,
    Busy => GVL_AXIS3.stTC_Home.Busy,
    Active => GVL_AXIS3.stTC_Home.Active,
    CommandAborted => GVL_AXIS3.stTC_Home.CmdAborted,
    Error => GVL_AXIS3.stTC_Home.Error,
    ErrorID => GVL_AXIS3.stTC_Home.ErrorID); // MC_Home
GVL_AXIS3.stTC_Home.Done := GVL_AXIS3.fbTC_Home.Done;

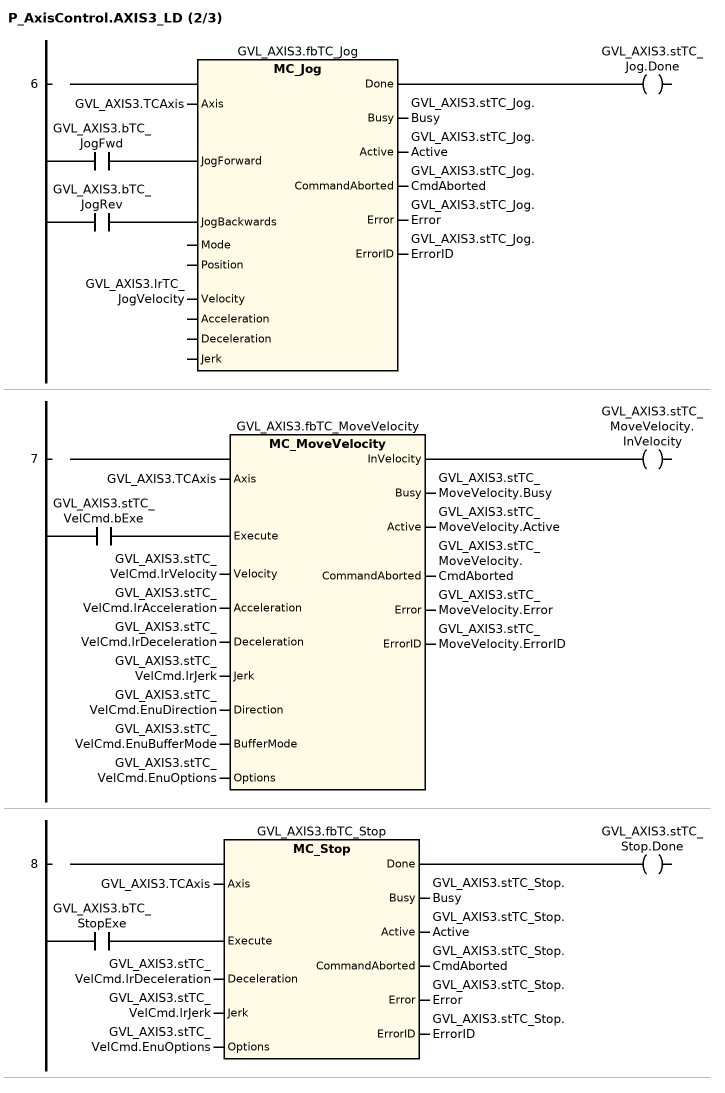
// NETWORK 6
GVL_AXIS3.fbTC_Jog(
    Axis := GVL_AXIS3.TCAxis,
    JogForward := GVL_AXIS3.bTC_JogFwd,
    JogBackwards := GVL_AXIS3.bTC_JogRev,
    Velocity := GVL_AXIS3.lrTC_JogVelocity,
    Busy => GVL_AXIS3.stTC_Jog.Busy,
    Active => GVL_AXIS3.stTC_Jog.Active,
    CommandAborted => GVL_AXIS3.stTC_Jog.CmdAborted,
    Error => GVL_AXIS3.stTC_Jog.Error,
    ErrorID => GVL_AXIS3.stTC_Jog.ErrorID); // MC_Jog
GVL_AXIS3.stTC_Jog.Done := GVL_AXIS3.fbTC_Jog.Done;

// NETWORK 7
GVL_AXIS3.fbTC_MoveVelocity(
    Axis := GVL_AXIS3.TCAxis,
    Execute := GVL_AXIS3.stTC_VelCmd.bExe,
    Velocity := GVL_AXIS3.stTC_VelCmd.lrVelocity,
    Acceleration := GVL_AXIS3.stTC_VelCmd.lrAcceleration,
    Deceleration := GVL_AXIS3.stTC_VelCmd.lrDeceleration,
    Jerk := GVL_AXIS3.stTC_VelCmd.lrJerk,
    Direction := GVL_AXIS3.stTC_VelCmd.EnuDirection,
    BufferMode := GVL_AXIS3.stTC_VelCmd.EnuBufferMode,
    Options := GVL_AXIS3.stTC_VelCmd.EnuOptions,
    Busy => GVL_AXIS3.stTC_MoveVelocity.Busy,
    Active => GVL_AXIS3.stTC_MoveVelocity.Active,
    CommandAborted => GVL_AXIS3.stTC_MoveVelocity.CmdAborted,
    Error => GVL_AXIS3.stTC_MoveVelocity.Error,
    ErrorID => GVL_AXIS3.stTC_MoveVelocity.ErrorID); // MC_MoveVelocity
GVL_AXIS3.stTC_MoveVelocity.InVelocity := GVL_AXIS3.fbTC_MoveVelocity.InVelocity;

// NETWORK 8
GVL_AXIS3.fbTC_Stop(
    Axis := GVL_AXIS3.TCAxis,
    Execute := GVL_AXIS3.bTC_StopExe,
    Deceleration := GVL_AXIS3.stTC_VelCmd.lrDeceleration,
    Jerk := GVL_AXIS3.stTC_VelCmd.lrJerk,
    Options := GVL_AXIS3.stTC_VelCmd.EnuOptions,
    Busy => GVL_AXIS3.stTC_Stop.Busy,
    Active => GVL_AXIS3.stTC_Stop.Active,
    CommandAborted => GVL_AXIS3.stTC_Stop.CmdAborted,
    Error => GVL_AXIS3.stTC_Stop.Error,
    ErrorID => GVL_AXIS3.stTC_Stop.ErrorID); // MC_Stop
GVL_AXIS3.stTC_Stop.Done := GVL_AXIS3.fbTC_Stop.Done;

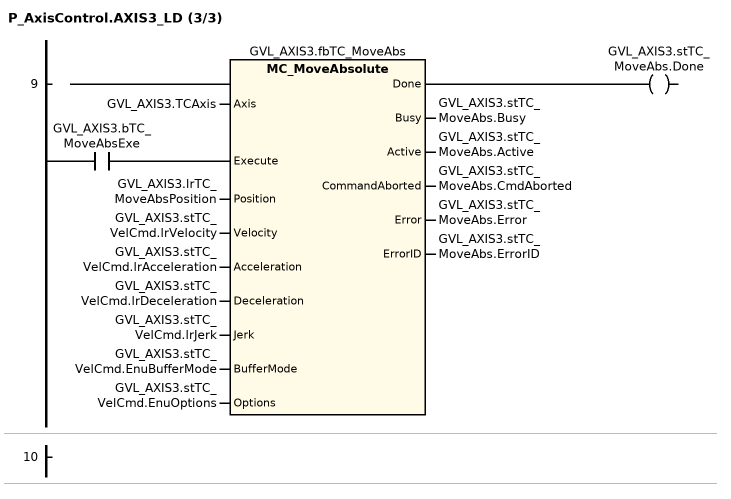
// NETWORK 9
GVL_AXIS3.fbTC_MoveAbs(
    Axis := GVL_AXIS3.TCAxis,
    Execute := GVL_AXIS3.bTC_MoveAbsExe,
    Position := GVL_AXIS3.lrTC_MoveAbsPosition,
    Velocity := GVL_AXIS3.stTC_VelCmd.lrVelocity,
    Acceleration := GVL_AXIS3.stTC_VelCmd.lrAcceleration,
    Deceleration := GVL_AXIS3.stTC_VelCmd.lrDeceleration,
    Jerk := GVL_AXIS3.stTC_VelCmd.lrJerk,
    BufferMode := GVL_AXIS3.stTC_VelCmd.EnuBufferMode,
    Options := GVL_AXIS3.stTC_VelCmd.EnuOptions,
    Busy => GVL_AXIS3.stTC_MoveAbs.Busy,
    Active => GVL_AXIS3.stTC_MoveAbs.Active,
    CommandAborted => GVL_AXIS3.stTC_MoveAbs.CmdAborted,
    Error => GVL_AXIS3.stTC_MoveAbs.Error,
    ErrorID => GVL_AXIS3.stTC_MoveAbs.ErrorID); // MC_MoveAbsolute
GVL_AXIS3.stTC_MoveAbs.Done := GVL_AXIS3.fbTC_MoveAbs.Done;

// NETWORK 10
END_METHOD

METHOD AXIS3_LD_Auto : BOOL
VAR_INPUT
END_VAR
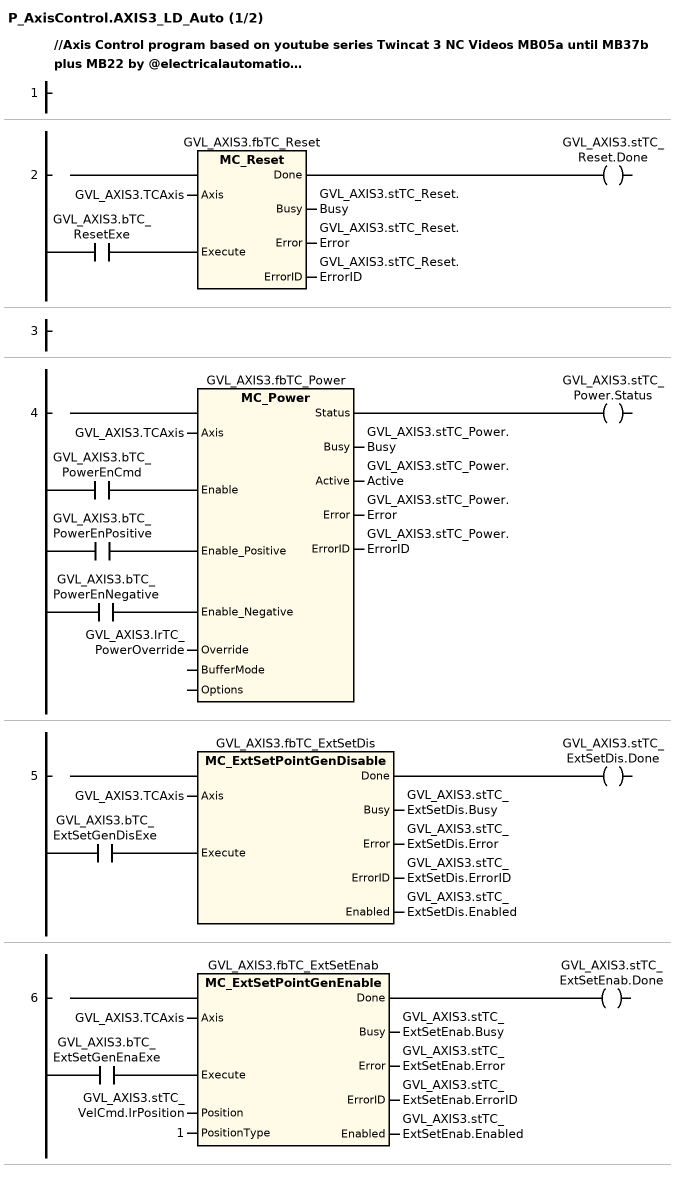
// NETWORK 1: //Axis Control program based on youtube series Twincat 3 NC Videos MB05a until MB37b plus MB22 by @electricalautomation https://www.youtube.com/watch?v=BxRAOdTks9I&list=PL762SfoJC-e8NbAUQ-H7a_TOdqrlBPCw4&index=25

// NETWORK 2
GVL_AXIS3.fbTC_Reset(
    Axis := GVL_AXIS3.TCAxis,
    Execute := GVL_AXIS3.bTC_ResetExe,
    Busy => GVL_AXIS3.stTC_Reset.Busy,
    Error => GVL_AXIS3.stTC_Reset.Error,
    ErrorID => GVL_AXIS3.stTC_Reset.ErrorID); // MC_Reset
GVL_AXIS3.stTC_Reset.Done := GVL_AXIS3.fbTC_Reset.Done;

// NETWORK 3

// NETWORK 4
GVL_AXIS3.fbTC_Power(
    Axis := GVL_AXIS3.TCAxis,
    Enable := GVL_AXIS3.bTC_PowerEnCmd,
    Enable_Positive := GVL_AXIS3.bTC_PowerEnPositive,
    Enable_Negative := GVL_AXIS3.bTC_PowerEnNegative,
    Override := GVL_AXIS3.lrTC_PowerOverride,
    Busy => GVL_AXIS3.stTC_Power.Busy,
    Active => GVL_AXIS3.stTC_Power.Active,
    Error => GVL_AXIS3.stTC_Power.Error,
    ErrorID => GVL_AXIS3.stTC_Power.ErrorID); // MC_Power
GVL_AXIS3.stTC_Power.Status := GVL_AXIS3.fbTC_Power.Status;

// NETWORK 5
GVL_AXIS3.fbTC_ExtSetDis(
    Axis := GVL_AXIS3.TCAxis,
    Execute := GVL_AXIS3.bTC_ExtSetGenDisExe,
    Busy => GVL_AXIS3.stTC_ExtSetDis.Busy,
    Error => GVL_AXIS3.stTC_ExtSetDis.Error,
    ErrorID => GVL_AXIS3.stTC_ExtSetDis.ErrorID,
    Enabled => GVL_AXIS3.stTC_ExtSetDis.Enabled); // MC_ExtSetPointGenDisable
GVL_AXIS3.stTC_ExtSetDis.Done := GVL_AXIS3.fbTC_ExtSetDis.Done;

// NETWORK 6
GVL_AXIS3.fbTC_ExtSetEnab(
    Axis := GVL_AXIS3.TCAxis,
    Execute := GVL_AXIS3.bTC_ExtSetGenEnaExe,
    Position := GVL_AXIS3.stTC_VelCmd.lrPosition,
    PositionType := 1,
    Busy => GVL_AXIS3.stTC_ExtSetEnab.Busy,
    Error => GVL_AXIS3.stTC_ExtSetEnab.Error,
    ErrorID => GVL_AXIS3.stTC_ExtSetEnab.ErrorID,
    Enabled => GVL_AXIS3.stTC_ExtSetEnab.Enabled); // MC_ExtSetPointGenEnable
GVL_AXIS3.stTC_ExtSetEnab.Done := GVL_AXIS3.fbTC_ExtSetEnab.Done;

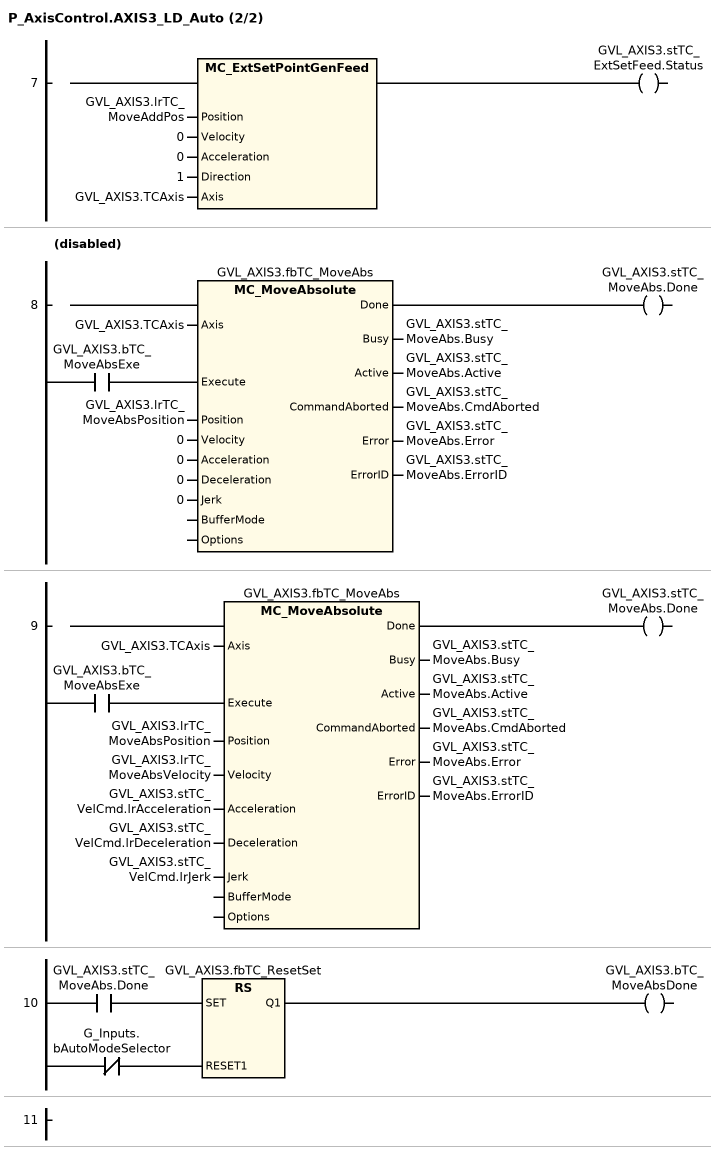
// NETWORK 7
GVL_AXIS3.stTC_ExtSetFeed.Status := MC_ExtSetPointGenFeed(Position := GVL_AXIS3.lrTC_MoveAddPos, Velocity := 0, Acceleration := 0, Direction := 1, Axis := GVL_AXIS3.TCAxis);

// NETWORK 8 (disabled)
// GVL_AXIS3.fbTC_MoveAbs(
//     Axis := GVL_AXIS3.TCAxis,
//     Execute := GVL_AXIS3.bTC_MoveAbsExe,
//     Position := GVL_AXIS3.lrTC_MoveAbsPosition,
//     Velocity := 0,
//     Acceleration := 0,
//     Deceleration := 0,
//     Jerk := 0,
//     Busy => GVL_AXIS3.stTC_MoveAbs.Busy,
//     Active => GVL_AXIS3.stTC_MoveAbs.Active,
//     CommandAborted => GVL_AXIS3.stTC_MoveAbs.CmdAborted,
//     Error => GVL_AXIS3.stTC_MoveAbs.Error,
//     ErrorID => GVL_AXIS3.stTC_MoveAbs.ErrorID); // MC_MoveAbsolute
// GVL_AXIS3.stTC_MoveAbs.Done := GVL_AXIS3.fbTC_MoveAbs.Done;

// NETWORK 9
GVL_AXIS3.fbTC_MoveAbs(
    Axis := GVL_AXIS3.TCAxis,
    Execute := GVL_AXIS3.bTC_MoveAbsExe,
    Position := GVL_AXIS3.lrTC_MoveAbsPosition,
    Velocity := GVL_AXIS3.lrTC_MoveAbsVelocity,
    Acceleration := GVL_AXIS3.stTC_VelCmd.lrAcceleration,
    Deceleration := GVL_AXIS3.stTC_VelCmd.lrDeceleration,
    Jerk := GVL_AXIS3.stTC_VelCmd.lrJerk,
    Busy => GVL_AXIS3.stTC_MoveAbs.Busy,
    Active => GVL_AXIS3.stTC_MoveAbs.Active,
    CommandAborted => GVL_AXIS3.stTC_MoveAbs.CmdAborted,
    Error => GVL_AXIS3.stTC_MoveAbs.Error,
    ErrorID => GVL_AXIS3.stTC_MoveAbs.ErrorID); // MC_MoveAbsolute
GVL_AXIS3.stTC_MoveAbs.Done := GVL_AXIS3.fbTC_MoveAbs.Done;

// NETWORK 10
GVL_AXIS3.fbTC_ResetSet(SET := GVL_AXIS3.stTC_MoveAbs.Done, RESET1 := NOT G_Inputs.bAutoModeSelector); // RS
GVL_AXIS3.bTC_MoveAbsDone := GVL_AXIS3.fbTC_ResetSet.Q1;

// NETWORK 11
END_METHOD

METHOD AXIS4_LD : BOOL
VAR_INPUT
END_VAR
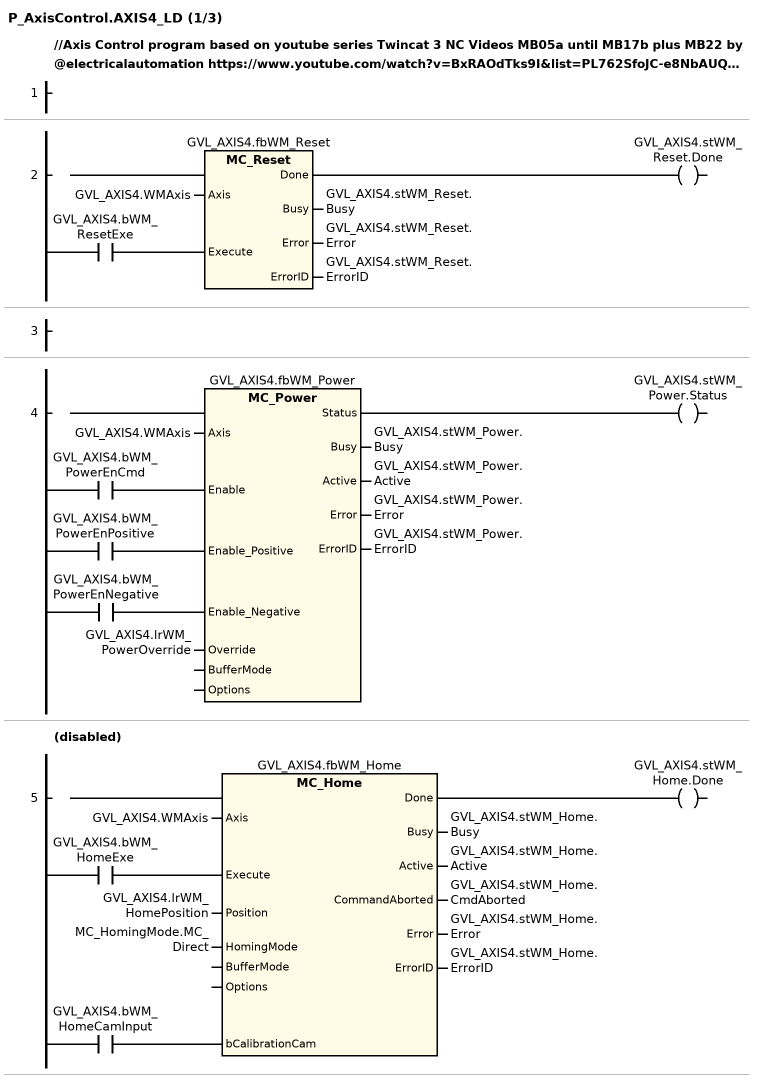
// NETWORK 1: //Axis Control program based on youtube series Twincat 3 NC Videos MB05a until MB17b plus MB22 by @electricalautomation https://www.youtube.com/watch?v=BxRAOdTks9I&list=PL762SfoJC-e8NbAUQ-H7a_TOdqrlBPCw4&index=25

// NETWORK 2
GVL_AXIS4.fbWM_Reset(
    Axis := GVL_AXIS4.WMAxis,
    Execute := GVL_AXIS4.bWM_ResetExe,
    Busy => GVL_AXIS4.stWM_Reset.Busy,
    Error => GVL_AXIS4.stWM_Reset.Error,
    ErrorID => GVL_AXIS4.stWM_Reset.ErrorID); // MC_Reset
GVL_AXIS4.stWM_Reset.Done := GVL_AXIS4.fbWM_Reset.Done;

// NETWORK 3

// NETWORK 4
GVL_AXIS4.fbWM_Power(
    Axis := GVL_AXIS4.WMAxis,
    Enable := GVL_AXIS4.bWM_PowerEnCmd,
    Enable_Positive := GVL_AXIS4.bWM_PowerEnPositive,
    Enable_Negative := GVL_AXIS4.bWM_PowerEnNegative,
    Override := GVL_AXIS4.lrWM_PowerOverride,
    Busy => GVL_AXIS4.stWM_Power.Busy,
    Active => GVL_AXIS4.stWM_Power.Active,
    Error => GVL_AXIS4.stWM_Power.Error,
    ErrorID => GVL_AXIS4.stWM_Power.ErrorID); // MC_Power
GVL_AXIS4.stWM_Power.Status := GVL_AXIS4.fbWM_Power.Status;

// NETWORK 5 (disabled)
// GVL_AXIS4.fbWM_Home(
//     Axis := GVL_AXIS4.WMAxis,
//     Execute := GVL_AXIS4.bWM_HomeExe,
//     Position := GVL_AXIS4.lrWM_HomePosition,
//     HomingMode := MC_HomingMode.MC_Direct,
//     bCalibrationCam := GVL_AXIS4.bWM_HomeCamInput,
//     Busy => GVL_AXIS4.stWM_Home.Busy,
//     Active => GVL_AXIS4.stWM_Home.Active,
//     CommandAborted => GVL_AXIS4.stWM_Home.CmdAborted,
//     Error => GVL_AXIS4.stWM_Home.Error,
//     ErrorID => GVL_AXIS4.stWM_Home.ErrorID); // MC_Home
// GVL_AXIS4.stWM_Home.Done := GVL_AXIS4.fbWM_Home.Done;

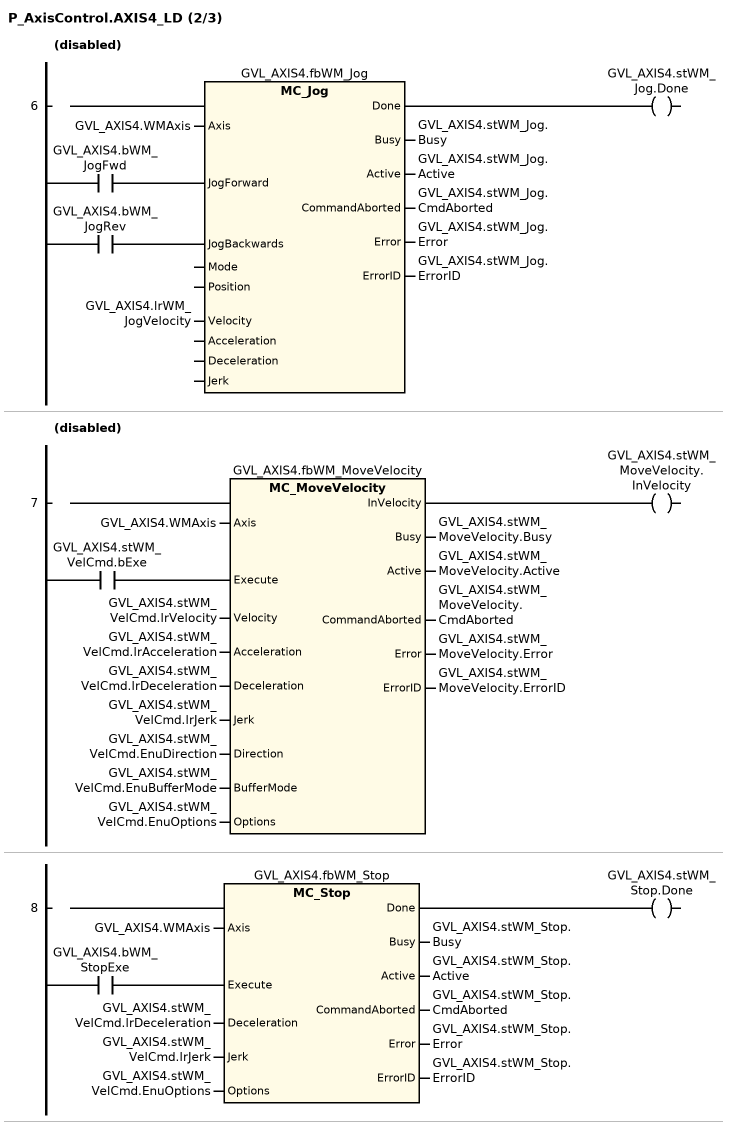
// NETWORK 6 (disabled)
// GVL_AXIS4.fbWM_Jog(
//     Axis := GVL_AXIS4.WMAxis,
//     JogForward := GVL_AXIS4.bWM_JogFwd,
//     JogBackwards := GVL_AXIS4.bWM_JogRev,
//     Velocity := GVL_AXIS4.lrWM_JogVelocity,
//     Busy => GVL_AXIS4.stWM_Jog.Busy,
//     Active => GVL_AXIS4.stWM_Jog.Active,
//     CommandAborted => GVL_AXIS4.stWM_Jog.CmdAborted,
//     Error => GVL_AXIS4.stWM_Jog.Error,
//     ErrorID => GVL_AXIS4.stWM_Jog.ErrorID); // MC_Jog
// GVL_AXIS4.stWM_Jog.Done := GVL_AXIS4.fbWM_Jog.Done;

// NETWORK 7 (disabled)
// GVL_AXIS4.fbWM_MoveVelocity(
//     Axis := GVL_AXIS4.WMAxis,
//     Execute := GVL_AXIS4.stWM_VelCmd.bExe,
//     Velocity := GVL_AXIS4.stWM_VelCmd.lrVelocity,
//     Acceleration := GVL_AXIS4.stWM_VelCmd.lrAcceleration,
//     Deceleration := GVL_AXIS4.stWM_VelCmd.lrDeceleration,
//     Jerk := GVL_AXIS4.stWM_VelCmd.lrJerk,
//     Direction := GVL_AXIS4.stWM_VelCmd.EnuDirection,
//     BufferMode := GVL_AXIS4.stWM_VelCmd.EnuBufferMode,
//     Options := GVL_AXIS4.stWM_VelCmd.EnuOptions,
//     Busy => GVL_AXIS4.stWM_MoveVelocity.Busy,
//     Active => GVL_AXIS4.stWM_MoveVelocity.Active,
//     CommandAborted => GVL_AXIS4.stWM_MoveVelocity.CmdAborted,
//     Error => GVL_AXIS4.stWM_MoveVelocity.Error,
//     ErrorID => GVL_AXIS4.stWM_MoveVelocity.ErrorID); // MC_MoveVelocity
// GVL_AXIS4.stWM_MoveVelocity.InVelocity := GVL_AXIS4.fbWM_MoveVelocity.InVelocity;

// NETWORK 8
GVL_AXIS4.fbWM_Stop(
    Axis := GVL_AXIS4.WMAxis,
    Execute := GVL_AXIS4.bWM_StopExe,
    Deceleration := GVL_AXIS4.stWM_VelCmd.lrDeceleration,
    Jerk := GVL_AXIS4.stWM_VelCmd.lrJerk,
    Options := GVL_AXIS4.stWM_VelCmd.EnuOptions,
    Busy => GVL_AXIS4.stWM_Stop.Busy,
    Active => GVL_AXIS4.stWM_Stop.Active,
    CommandAborted => GVL_AXIS4.stWM_Stop.CmdAborted,
    Error => GVL_AXIS4.stWM_Stop.Error,
    ErrorID => GVL_AXIS4.stWM_Stop.ErrorID); // MC_Stop
GVL_AXIS4.stWM_Stop.Done := GVL_AXIS4.fbWM_Stop.Done;

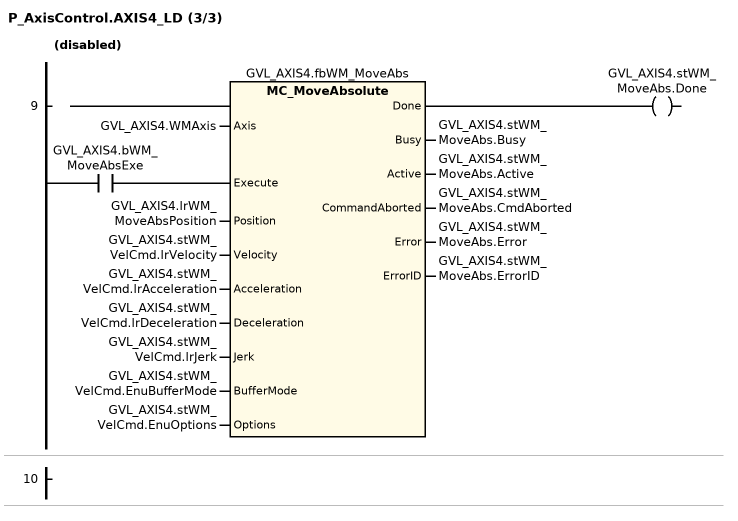
// NETWORK 9 (disabled)
// GVL_AXIS4.fbWM_MoveAbs(
//     Axis := GVL_AXIS4.WMAxis,
//     Execute := GVL_AXIS4.bWM_MoveAbsExe,
//     Position := GVL_AXIS4.lrWM_MoveAbsPosition,
//     Velocity := GVL_AXIS4.stWM_VelCmd.lrVelocity,
//     Acceleration := GVL_AXIS4.stWM_VelCmd.lrAcceleration,
//     Deceleration := GVL_AXIS4.stWM_VelCmd.lrDeceleration,
//     Jerk := GVL_AXIS4.stWM_VelCmd.lrJerk,
//     BufferMode := GVL_AXIS4.stWM_VelCmd.EnuBufferMode,
//     Options := GVL_AXIS4.stWM_VelCmd.EnuOptions,
//     Busy => GVL_AXIS4.stWM_MoveAbs.Busy,
//     Active => GVL_AXIS4.stWM_MoveAbs.Active,
//     CommandAborted => GVL_AXIS4.stWM_MoveAbs.CmdAborted,
//     Error => GVL_AXIS4.stWM_MoveAbs.Error,
//     ErrorID => GVL_AXIS4.stWM_MoveAbs.ErrorID); // MC_MoveAbsolute
// GVL_AXIS4.stWM_MoveAbs.Done := GVL_AXIS4.fbWM_MoveAbs.Done;

// NETWORK 10
END_METHOD

METHOD AXIS4_LD_Auto : BOOL
VAR_INPUT
END_VAR
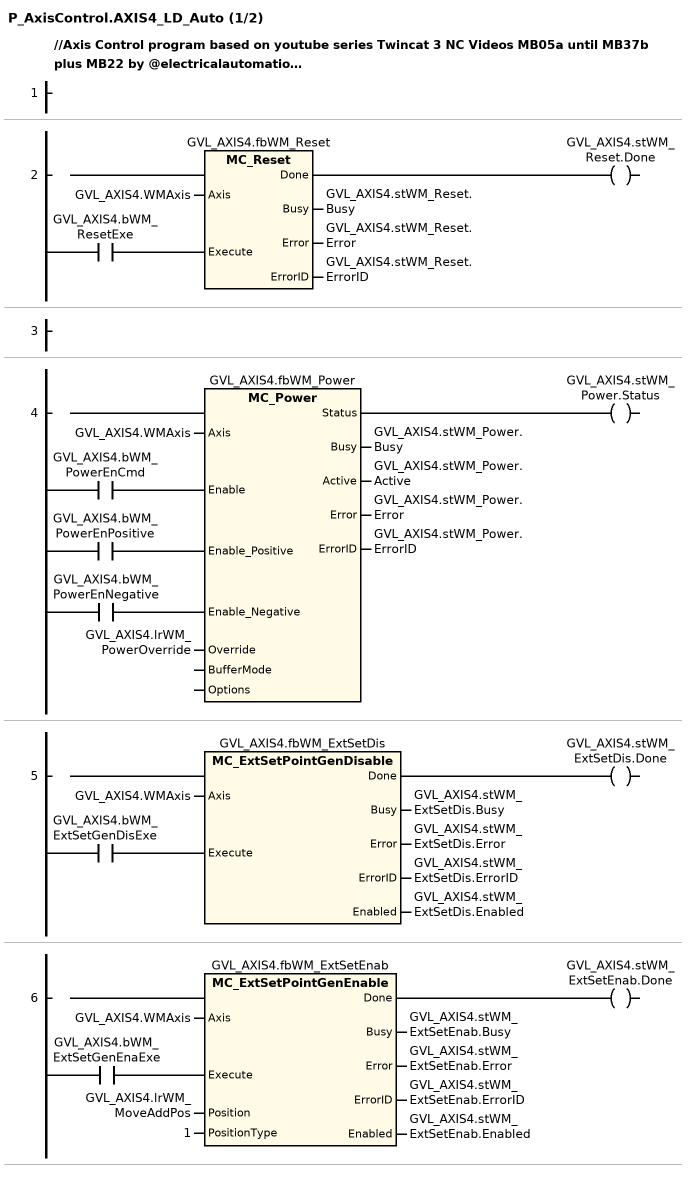
// NETWORK 1: //Axis Control program based on youtube series Twincat 3 NC Videos MB05a until MB37b plus MB22 by @electricalautomation https://www.youtube.com/waWMh?v=BxRAOdTks9I&list=PL762SfoJC-e8NbAUQ-H7a_TOdqrlBPCw4&index=25

// NETWORK 2
GVL_AXIS4.fbWM_Reset(
    Axis := GVL_AXIS4.WMAxis,
    Execute := GVL_AXIS4.bWM_ResetExe,
    Busy => GVL_AXIS4.stWM_Reset.Busy,
    Error => GVL_AXIS4.stWM_Reset.Error,
    ErrorID => GVL_AXIS4.stWM_Reset.ErrorID); // MC_Reset
GVL_AXIS4.stWM_Reset.Done := GVL_AXIS4.fbWM_Reset.Done;

// NETWORK 3

// NETWORK 4
GVL_AXIS4.fbWM_Power(
    Axis := GVL_AXIS4.WMAxis,
    Enable := GVL_AXIS4.bWM_PowerEnCmd,
    Enable_Positive := GVL_AXIS4.bWM_PowerEnPositive,
    Enable_Negative := GVL_AXIS4.bWM_PowerEnNegative,
    Override := GVL_AXIS4.lrWM_PowerOverride,
    Busy => GVL_AXIS4.stWM_Power.Busy,
    Active => GVL_AXIS4.stWM_Power.Active,
    Error => GVL_AXIS4.stWM_Power.Error,
    ErrorID => GVL_AXIS4.stWM_Power.ErrorID); // MC_Power
GVL_AXIS4.stWM_Power.Status := GVL_AXIS4.fbWM_Power.Status;

// NETWORK 5
GVL_AXIS4.fbWM_ExtSetDis(
    Axis := GVL_AXIS4.WMAxis,
    Execute := GVL_AXIS4.bWM_ExtSetGenDisExe,
    Busy => GVL_AXIS4.stWM_ExtSetDis.Busy,
    Error => GVL_AXIS4.stWM_ExtSetDis.Error,
    ErrorID => GVL_AXIS4.stWM_ExtSetDis.ErrorID,
    Enabled => GVL_AXIS4.stWM_ExtSetDis.Enabled); // MC_ExtSetPointGenDisable
GVL_AXIS4.stWM_ExtSetDis.Done := GVL_AXIS4.fbWM_ExtSetDis.Done;

// NETWORK 6
GVL_AXIS4.fbWM_ExtSetEnab(
    Axis := GVL_AXIS4.WMAxis,
    Execute := GVL_AXIS4.bWM_ExtSetGenEnaExe,
    Position := GVL_AXIS4.lrWM_MoveAddPos,
    PositionType := 1,
    Busy => GVL_AXIS4.stWM_ExtSetEnab.Busy,
    Error => GVL_AXIS4.stWM_ExtSetEnab.Error,
    ErrorID => GVL_AXIS4.stWM_ExtSetEnab.ErrorID,
    Enabled => GVL_AXIS4.stWM_ExtSetEnab.Enabled); // MC_ExtSetPointGenEnable
GVL_AXIS4.stWM_ExtSetEnab.Done := GVL_AXIS4.fbWM_ExtSetEnab.Done;

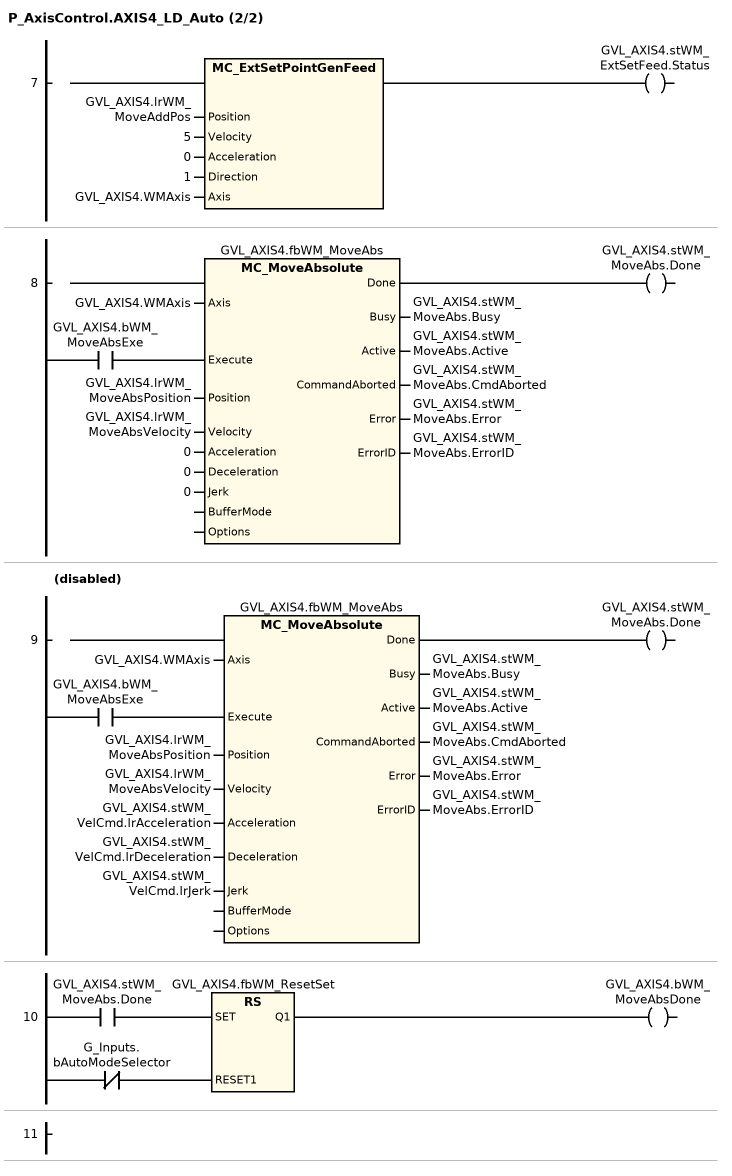
// NETWORK 7
GVL_AXIS4.stWM_ExtSetFeed.Status := MC_ExtSetPointGenFeed(Position := GVL_AXIS4.lrWM_MoveAddPos, Velocity := 5, Acceleration := 0, Direction := 1, Axis := GVL_AXIS4.WMAxis);

// NETWORK 8
GVL_AXIS4.fbWM_MoveAbs(
    Axis := GVL_AXIS4.WMAxis,
    Execute := GVL_AXIS4.bWM_MoveAbsExe,
    Position := GVL_AXIS4.lrWM_MoveAbsPosition,
    Velocity := GVL_AXIS4.lrWM_MoveAbsVelocity,
    Acceleration := 0,
    Deceleration := 0,
    Jerk := 0,
    Busy => GVL_AXIS4.stWM_MoveAbs.Busy,
    Active => GVL_AXIS4.stWM_MoveAbs.Active,
    CommandAborted => GVL_AXIS4.stWM_MoveAbs.CmdAborted,
    Error => GVL_AXIS4.stWM_MoveAbs.Error,
    ErrorID => GVL_AXIS4.stWM_MoveAbs.ErrorID); // MC_MoveAbsolute
GVL_AXIS4.stWM_MoveAbs.Done := GVL_AXIS4.fbWM_MoveAbs.Done;

// NETWORK 9 (disabled)
// GVL_AXIS4.fbWM_MoveAbs(
//     Axis := GVL_AXIS4.WMAxis,
//     Execute := GVL_AXIS4.bWM_MoveAbsExe,
//     Position := GVL_AXIS4.lrWM_MoveAbsPosition,
//     Velocity := GVL_AXIS4.lrWM_MoveAbsVelocity,
//     Acceleration := GVL_AXIS4.stWM_VelCmd.lrAcceleration,
//     Deceleration := GVL_AXIS4.stWM_VelCmd.lrDeceleration,
//     Jerk := GVL_AXIS4.stWM_VelCmd.lrJerk,
//     Busy => GVL_AXIS4.stWM_MoveAbs.Busy,
//     Active => GVL_AXIS4.stWM_MoveAbs.Active,
//     CommandAborted => GVL_AXIS4.stWM_MoveAbs.CmdAborted,
//     Error => GVL_AXIS4.stWM_MoveAbs.Error,
//     ErrorID => GVL_AXIS4.stWM_MoveAbs.ErrorID); // MC_MoveAbsolute
// GVL_AXIS4.stWM_MoveAbs.Done := GVL_AXIS4.fbWM_MoveAbs.Done;

// NETWORK 10
GVL_AXIS4.fbWM_ResetSet(SET := GVL_AXIS4.stWM_MoveAbs.Done, RESET1 := NOT G_Inputs.bAutoModeSelector); // RS
GVL_AXIS4.bWM_MoveAbsDone := GVL_AXIS4.fbWM_ResetSet.Q1;

// NETWORK 11
END_METHOD

METHOD Manual_mode : BOOL
VAR_INPUT
END_VAR
//Axis 1 Main arm actuator
AXIS1_LD();

GVL_AXIS1.bBC_ResetExe := FALSE;

GVL_AXIS1.stBC_VelCmd.EnuDirection := MC_Undefined_Direction;

GVL_AXIS1.stBC_VelCmd.bExe := FALSE;

GVL_AXIS1.bBC_PowerEnCmd := G_Inputs.bManualModeSelector;

IF G_Sensors.fJoystickLeftNormalizedX  > 0 AND G_Inputs.bJoystickLeftEnable THEN
	GVL_AXIS1.bBC_PowerEnNegative := TRUE;
	GVL_AXIS1.stBC_VelCmd.EnuDirection := MC_Negative_Direction;
	GVL_AXIS1.lrBC_PowerOverride := ABS(G_Sensors.fJoystickLeftNormalizedX) * 100;	
	GVL_AXIS1.stBC_VelCmd.bExe := TRUE;
ELSIF G_Sensors.fJoystickLeftNormalizedX < 0 AND G_Inputs.bJoystickLeftEnable THEN
	GVL_AXIS1.bBC_PowerEnPositive := TRUE;
	GVL_AXIS1.stBC_VelCmd.EnuDirection := MC_Positive_Direction;
	GVL_AXIS1.lrBC_PowerOverride := ABS(G_Sensors.fJoystickLeftNormalizedX) * 100;	
	GVL_AXIS1.stBC_VelCmd.bExe := TRUE;
ELSE
	 GVL_AXIS1.lrBC_PowerOverride := 0;
	 GVL_AXIS1.stBC_VelCmd.bExe := FALSE;
	 GVL_AXIS1.bBC_PowerEnNegative := FALSE;
	 GVL_AXIS1.bBC_PowerEnPositive := FALSE;
END_IF

GVL_AXIS1.bBC_ResetExe := TRUE;


//Axis 2 Slew joint actuator
AXIS2_LD();

GVL_AXIS2.bSJ_ResetExe := FALSE;

GVL_AXIS2.stSJ_VelCmd.EnuDirection := MC_Undefined_Direction;

GVL_AXIS2.stSJ_VelCmd.bExe := FALSE;

GVL_AXIS2.bSJ_PowerEnCmd := G_Inputs.bManualModeSelector;

IF G_Sensors.fJoystickRightNormalizedX  > 0 AND G_Inputs.bJoystickRightEnable THEN
	GVL_AXIS2.bSJ_PowerEnPositive := TRUE;
	GVL_AXIS2.stSJ_VelCmd.EnuDirection := MC_Positive_Direction;
	GVL_AXIS2.lrSJ_PowerOverride := ABS(G_Sensors.fJoystickRightNormalizedX) * 100;	
	GVL_AXIS2.stSJ_VelCmd.bExe := TRUE;
ELSIF G_Sensors.fJoystickRightNormalizedX < 0 AND G_Inputs.bJoystickRightEnable THEN
	GVL_AXIS2.bSJ_PowerEnNegative := TRUE;
	GVL_AXIS2.stSJ_VelCmd.EnuDirection := MC_Negative_Direction;
	GVL_AXIS2.lrSJ_PowerOverride := ABS(G_Sensors.fJoystickRightNormalizedX) * 100;	
	GVL_AXIS2.stSJ_VelCmd.bExe := TRUE;
ELSE
	 GVL_AXIS2.lrSJ_PowerOverride := 0;
	 GVL_AXIS2.stSJ_VelCmd.bExe := FALSE;
	 GVL_AXIS2.bSJ_PowerEnNegative := FALSE;
	 GVL_AXIS2.bSJ_PowerEnPositive := FALSE;
END_IF

GVL_AXIS2.bSJ_ResetExe := TRUE;


//Axis 3 Knuckle arm actuator
AXIS3_LD();

GVL_AXIS3.bTC_ResetExe := FALSE;

GVL_AXIS3.stTC_VelCmd.EnuDirection := MC_Undefined_Direction;

GVL_AXIS3.stTC_VelCmd.bExe := FALSE;

GVL_AXIS3.bTC_PowerEnCmd := G_Inputs.bManualModeSelector;

IF G_Sensors.fJoystickLeftNormalizedY  > 0 AND G_Inputs.bJoystickLeftEnable THEN
	GVL_AXIS3.bTC_PowerEnPositive := TRUE;
	GVL_AXIS3.stTC_VelCmd.EnuDirection := MC_Positive_Direction;
	GVL_AXIS3.lrTC_PowerOverride := ABS(G_Sensors.fJoystickLeftNormalizedY) * 100;	
	GVL_AXIS3.stTC_VelCmd.bExe := TRUE;
ELSIF G_Sensors.fJoystickLeftNormalizedY < 0 AND G_Inputs.bJoystickLeftEnable THEN
	GVL_AXIS3.bTC_PowerEnNegative := TRUE;
	GVL_AXIS3.stTC_VelCmd.EnuDirection := MC_Negative_Direction;
	GVL_AXIS3.lrTC_PowerOverride := ABS(G_Sensors.fJoystickLeftNormalizedY) * 100;	
	GVL_AXIS3.stTC_VelCmd.bExe := TRUE;
ELSE
	 GVL_AXIS3.lrTC_PowerOverride := 0;
	 GVL_AXIS3.stTC_VelCmd.bExe := FALSE;
	 GVL_AXIS3.bTC_PowerEnNegative := FALSE;
	 GVL_AXIS3.bTC_PowerEnPositive := FALSE;
END_IF

GVL_AXIS3.bTC_ResetExe := TRUE;

(*
AXIS3_LD();

GVL_AXIS3.bTC_ResetExe := G_Inputs.bJoystickLeftEnable;

GVL_AXIS3.EnuMoveVelDirection := G_Sensors.MCDirectionAxis3;

GVL_AXIS3.bTC_PowerEnCmd := G_Inputs.bManualModeSelector;
GVL_AXIS3.bTC_PowerEnNegative := G_Inputs.bManualModeSelector;
GVL_AXIS3.bTC_PowerEnPositive := G_Inputs.bManualModeSelector;


// Velocity control
IF G_Sensors.fJoystickLeftNormalizedY  > 0.01 AND G_Inputs.bJoystickLeftEnable THEN
	GVL_AXIS3.stTC_VelCmd.EnuDirection := MC_Positive_Direction;
	GVL_AXIS3.lrTC_PowerOverride := ABS(G_Sensors.fJoystickLeftNormalizedY) * 100;	
	GVL_AXIS3.stTC_VelCmd.bExe := TRUE;
ELSIF G_Sensors.fJoystickLeftNormalizedY < 0.01 AND G_Inputs.bJoystickLeftEnable THEN
	GVL_AXIS3.stTC_VelCmd.EnuDirection := MC_Negative_Direction;
	GVL_AXIS3.lrTC_PowerOverride := ABS(G_Sensors.fJoystickLeftNormalizedY) * 100;	
	GVL_AXIS3.stTC_VelCmd.bExe := TRUE;
ELSE
	 GVL_AXIS3.lrTC_PowerOverride := 0;
	 //GVL_AXIS3.stTC_VelCmd.EnuDirection := MC_Current_Direction;
	 GVL_AXIS3.stTC_VelCmd.bExe := FALSE;
END_IF
*)

(*
AXIS4_LD();

GVL_AXIS4.bWM_ResetExe := G_Inputs.bJoystickRightEnable;

GVL_AXIS4.EnuMoveVelDirection := G_Sensors.MCDirectionAxis4;

GVL_AXIS4.bWM_PowerEnCmd := G_Inputs.bManualModeSelector;
GVL_AXIS4.bWM_PowerEnNegative := G_Inputs.bManualModeSelector;
GVL_AXIS4.bWM_PowerEnPositive := G_Inputs.bManualModeSelector;


// Velocity control
IF G_Sensors.fJoystickLeftNormalizedY  > 0 AND G_Inputs.bJoystickRightEnable THEN
	GVL_AXIS4.lrWM_PowerOverride := ABS(G_Sensors.fJoystickRightNormalizedY) * 100;
	GVL_AXIS4.stWM_VelCmd.EnuDirection := MC_Positive_Direction;
	GVL_AXIS4.stWM_VelCmd.bExe := TRUE;
ELSIF G_Sensors.fJoystickLeftNormalizedY < 0 AND G_Inputs.bJoystickLeftEnable THEN
	GVL_AXIS4.lrWM_PowerOverride := ABS(G_Sensors.fJoystickLeftNormalizedY) * 100;
	GVL_AXIS4.stWM_VelCmd.EnuDirection := MC_Negative_Direction;
	GVL_AXIS4.stWM_VelCmd.bExe := TRUE;
ELSE
	 GVL_AXIS4.lrWM_PowerOverride := 0;
	 GVL_AXIS4.stWM_VelCmd.EnuDirection := MC_Current_Direction;
	 GVL_AXIS4.stWM_VelCmd.bExe := FALSE;
END_IF
*)

//Axis 4 Winch motor actuator
AXIS4_LD();

GVL_AXIS4.bWM_ResetExe := FALSE;

GVL_AXIS4.stWM_VelCmd.EnuDirection := MC_Undefined_Direction;

GVL_AXIS4.stWM_VelCmd.bExe := FALSE;

GVL_AXIS4.bWM_PowerEnCmd := G_Inputs.bManualModeSelector;

IF G_Sensors.fJoystickRightNormalizedY  > 0 AND G_Inputs.bJoystickRightEnable THEN
	GVL_AXIS4.bWM_PowerEnNegative := TRUE;
	GVL_AXIS4.stWM_VelCmd.EnuDirection := MC_Negative_Direction;
	GVL_AXIS4.lrWM_PowerOverride := ABS(G_Sensors.fJoystickRightNormalizedY) * 100;	
	GVL_AXIS4.stWM_VelCmd.bExe := TRUE;
ELSIF G_Sensors.fJoystickRightNormalizedY < 0 AND G_Inputs.bJoystickRightEnable THEN
	GVL_AXIS4.bWM_PowerEnPositive := TRUE;
	GVL_AXIS4.stWM_VelCmd.EnuDirection := MC_Positive_Direction;
	GVL_AXIS4.lrWM_PowerOverride := ABS(G_Sensors.fJoystickRightNormalizedY) * 100;	
	GVL_AXIS4.stWM_VelCmd.bExe := TRUE;
ELSE
	 GVL_AXIS4.lrWM_PowerOverride := 0;
	 GVL_AXIS4.stWM_VelCmd.bExe := FALSE;
	 GVL_AXIS4.bWM_PowerEnNegative := FALSE;
	 GVL_AXIS4.bWM_PowerEnPositive := FALSE;
END_IF

GVL_AXIS4.bWM_ResetExe := TRUE;
END_METHOD

END_PROGRAM

// ---- AXIS CONTROL/P_AxisControl_1.TcPOU
PROGRAM P_AxisControl_1
VAR
END_VAR

//Axis Control program based on youtube series Twincat 3 NC Videos MB05a until MB17b plus MB22 by @electricalautomation https://www.youtube.com/watch?v=BxRAOdTks9I&list=PL762SfoJC-e8NbAUQ-H7a_TOdqrlBPCw4&index=25

AXIS1_LD();

GVL_AXIS1.bBC_ResetExe := G_Inputs.bJoystickLeftEnable OR G_Inputs.bAutoModeSelector;

GVL_AXIS1.EnuMoveVelDirection := G_Sensors.MCDirectionAxis1;

GVL_AXIS1.bBC_PowerEnCmd := G_Inputs.bManualModeSelector OR G_Inputs.bAutoModeSelector;
GVL_AXIS1.bBC_PowerEnNegative := G_Inputs.bManualModeSelector OR G_Inputs.bAutoModeSelector;
GVL_AXIS1.bBC_PowerEnPositive := G_Inputs.bManualModeSelector OR G_Inputs.bAutoModeSelector;

//GVL_AXIS1.lrBC_PowerOverride := 50;

GVL_AXIS1.lrBC_MoveAddPos := GVL_InverseKinematics.fStrokeActuatorMainInverse*1000; //Position in mm
GVL_AXIS1.stBC_VelCmd.lrPosition := GVL_InverseKinematics.fStrokeActuatorMainInverse*1000; //Position in mm

GVL_AXIS1.lrBC_MoveContAbsEndVel := 0;


// Jog control

(*
IF G_Sensors.fJoystickLeftNormalizedX  > 0 AND G_Inputs.bJoystickLeftEnable THEN
	GVL_AXIS1.bBC_JogRev := TRUE;
ELSIF G_Sensors.fJoystickLeftNormalizedX < 0 AND G_Inputs.bJoystickLeftEnable THEN
	GVL_AXIS1.bBC_JogFwd := TRUE;
ELSE
	 GVL_AXIS1.bBC_JogFwd := FALSE;
	 GVL_AXIS1.bBC_JogRev := FALSE;
END_IF

*)

//Position control
IF G_Inputs.bAutoModeSelector AND G_Inputs.bJoystickLeftEnable THEN
	GVL_AXIS1.bBC_ExtSetGenDisExe := FALSE;
	GVL_AXIS1.bBC_ExtSetGenEnaExe := TRUE;
ELSE
	GVL_AXIS1.bBC_ExtSetGenDisExe := TRUE;
	GVL_AXIS1.bBC_ExtSetGenEnaExe := FALSE;
END_IF

GVL_AXIS1.lrBC_PosError := GVL_InverseKinematics.fStrokeActuatorMainInverse*1000 - GVL_AXIS1.lrBC_ActPos;

IF GVL_AXIS1.lrBC_PosError > 0 THEN
	GVL_AXIS1.fBC_ExtSetFeedDirection := 1;
ELSIF GVL_AXIS1.lrBC_PosError < 0 THEN
	GVL_AXIS1.fBC_ExtSetFeedDirection := -1;
ELSE
	GVL_AXIS1.fBC_ExtSetFeedDirection := 0;
END_IF

// Manual velocity control
IF G_Sensors.fJoystickLeftNormalizedX  >= 0 AND G_Inputs.bJoystickLeftEnable AND G_Inputs.bManualModeSelector THEN
	GVL_AXIS1.lrBC_PowerOverride := ABS(G_Sensors.fJoystickLeftNormalizedX) * 100;
	GVL_AXIS1.stBC_VelCmd.EnuDirection := MC_Positive_Direction;
	GVL_AXIS1.stBC_VelCmd.bExe := TRUE;
ELSIF G_Sensors.fJoystickLeftNormalizedX < 0 AND G_Inputs.bJoystickLeftEnable AND G_Inputs.bManualModeSelector THEN
	GVL_AXIS1.lrBC_PowerOverride := ABS(G_Sensors.fJoystickLeftNormalizedX) * 100;
	GVL_AXIS1.stBC_VelCmd.EnuDirection := MC_Negative_Direction;
	GVL_AXIS1.stBC_VelCmd.bExe := TRUE;
ELSE
	 GVL_AXIS1.lrBC_PowerOverride := 0;
	 //GVL_AXIS1.stBC_VelCmd.EnuDirection := MC_Current_Direction;
	 GVL_AXIS1.stBC_VelCmd.bExe := FALSE;
	 GVL_AXIS1.bBC_StopExe := TRUE;
END_IF


(*
// Automatic position control

IF G_Inputs.bAutoModeSelector THEN
	GVL_AXIS1.lrBC_PowerOverride := 10;
	//GVL_AXIS1.stBC_VelCmd.EnuDirection := MC_Positive_Direction;
	GVL_AXIS1.stBC_VelCmd.bExe := TRUE;
	GVL_AXIS1.bBC_MoveAbsExe := TRUE;
ELSE
	 GVL_AXIS1.lrBC_PowerOverride := 0;
	 //GVL_AXIS1.stBC_VelCmd.EnuDirection := MC_Current_Direction;
	 GVL_AXIS1.stBC_VelCmd.bExe := FALSE;
END_IF
*)

AXIS2_LD();

GVL_AXIS2.bSJ_ResetExe := G_Inputs.bJoystickRightEnable;

GVL_AXIS2.EnuMoveVelDirection := G_Sensors.MCDirectionAxis2;

GVL_AXIS2.bSJ_PowerEnCmd := G_Inputs.bManualModeSelector;
GVL_AXIS2.bSJ_PowerEnNegative := G_Inputs.bManualModeSelector;
GVL_AXIS2.bSJ_PowerEnPositive := G_Inputs.bManualModeSelector;

GVL_AXIS2.lrSJ_JogVelocity := 100;


// Velocity control
IF G_Sensors.fJoystickRightNormalizedX  > 0 AND G_Inputs.bJoystickRightEnable THEN
	GVL_AXIS2.lrSJ_PowerOverride := ABS(G_Sensors.fJoystickRightNormalizedX) * 100;
	GVL_AXIS2.stSJ_VelCmd.EnuDirection := MC_Positive_Direction;
	GVL_AXIS2.stSJ_VelCmd.bExe := TRUE;
ELSIF G_Sensors.fJoystickRightNormalizedX < 0 AND G_Inputs.bJoystickRightEnable THEN
	GVL_AXIS2.lrSJ_PowerOverride := ABS(G_Sensors.fJoystickRightNormalizedX) * 100;
	GVL_AXIS2.stSJ_VelCmd.EnuDirection := MC_Negative_Direction;
	GVL_AXIS2.stSJ_VelCmd.bExe := TRUE;
ELSE
	 GVL_AXIS2.lrSJ_PowerOverride := 0;
	 //GVL_AXIS2.stSJ_VelCmd.EnuDirection := MC_Current_Direction;
	 GVL_AXIS2.stSJ_VelCmd.bExe := FALSE;
END_IF


AXIS3_LD();

GVL_AXIS3.bTC_ResetExe := G_Inputs.bJoystickLeftEnable;

GVL_AXIS3.EnuMoveVelDirection := G_Sensors.MCDirectionAxis3;

GVL_AXIS3.bTC_PowerEnCmd := G_Inputs.bManualModeSelector;
GVL_AXIS3.bTC_PowerEnNegative := G_Inputs.bManualModeSelector;
GVL_AXIS3.bTC_PowerEnPositive := G_Inputs.bManualModeSelector;

GVL_AXIS3.lrTC_JogVelocity := 100;


// Velocity control
IF G_Sensors.fJoystickLeftNormalizedY  > 0 AND G_Inputs.bJoystickLeftEnable THEN
	GVL_AXIS3.lrTC_PowerOverride := ABS(G_Sensors.fJoystickLeftNormalizedY) * 100;
	GVL_AXIS3.stTC_VelCmd.EnuDirection := MC_Positive_Direction;
	GVL_AXIS3.stTC_VelCmd.bExe := TRUE;
ELSIF G_Sensors.fJoystickLeftNormalizedY < 0 AND G_Inputs.bJoystickLeftEnable THEN
	GVL_AXIS3.lrTC_PowerOverride := ABS(G_Sensors.fJoystickLeftNormalizedY) * 100;
	GVL_AXIS3.stTC_VelCmd.EnuDirection := MC_Negative_Direction;
	GVL_AXIS3.stTC_VelCmd.bExe := TRUE;
ELSE
	 GVL_AXIS3.lrTC_PowerOverride := 0;
	 //GVL_AXIS3.stTC_VelCmd.EnuDirection := MC_Current_Direction;
	 GVL_AXIS3.stTC_VelCmd.bExe := FALSE;
END_IF

(*
AXIS4_LD();

//Safety
GVL_Safety_AXIS4.bSafetyRestart := GVL_AXIS4.bInAckSignal;
GVL_Safety_AXIS4.bErrorAck		:= GVL_AXIS4.bInAckSignal;
GVL_Safety_AXIS4.bSafetyRun		:= TRUE;

//
GVL_AXIS4.bWM_ResetExe := G_Inputs.bJoystickLeftEnable;

GVL_AXIS4.EnuMoveVelDirection := G_Sensors.MCDirectionAxis4;

GVL_AXIS4.bWM_PowerEnCmd := G_Inputs.bManualModeSelector;
GVL_AXIS4.bWM_PowerEnNegative := G_Inputs.bManualModeSelector;
GVL_AXIS4.bWM_PowerEnPositive := G_Inputs.bManualModeSelector;

GVL_AXIS4.lrWM_JogVelocity := 100;
//GVL_AXIS4.lrWM_PowerOverride := 50;


// Velocity control
IF G_Sensors.fJoystickLeftNormalizedY  > 0 AND G_Inputs.bJoystickLeftEnable THEN
	GVL_AXIS4.lrWM_PowerOverride := ABS(G_Sensors.fJoystickLeftNormalizedY) * 100;
	GVL_AXIS4.stWM_VelCmd.EnuDirection := MC_Positive_Direction;
	GVL_AXIS4.stWM_VelCmd.bExe := TRUE;
ELSIF G_Sensors.fJoystickLeftNormalizedY < 0 AND G_Inputs.bJoystickLeftEnable THEN
	GVL_AXIS4.lrWM_PowerOverride := ABS(G_Sensors.fJoystickLeftNormalizedY) * 100;
	GVL_AXIS4.stWM_VelCmd.EnuDirection := MC_Negative_Direction;
	GVL_AXIS4.stWM_VelCmd.bExe := TRUE;
ELSE
	 GVL_AXIS4.lrWM_PowerOverride := 0;
	 GVL_AXIS4.stWM_VelCmd.EnuDirection := MC_Current_Direction;
	 GVL_AXIS4.stWM_VelCmd.bExe := FALSE;
END_IF
*)

METHOD Auto_mode : BOOL
VAR_INPUT
END_VAR
END_METHOD

METHOD AXIS1_LD : BOOL
VAR_INPUT
END_VAR
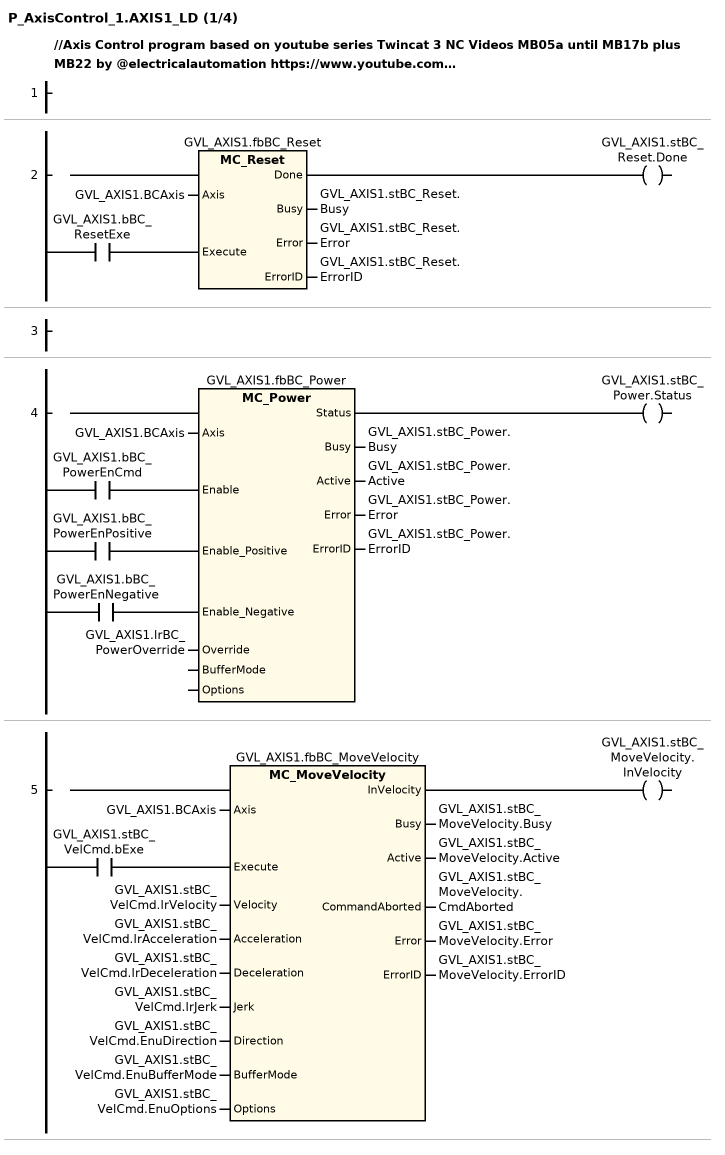
// NETWORK 1: //Axis Control program based on youtube series Twincat 3 NC Videos MB05a until MB17b plus MB22 by @electricalautomation https://www.youtube.com/watch?v=BxRAOdTks9I&list=PL762SfoJC-e8NbAUQ-H7a_TOdqrlBPCw4&index=25

// NETWORK 2
GVL_AXIS1.fbBC_Reset(
    Axis := GVL_AXIS1.BCAxis,
    Execute := GVL_AXIS1.bBC_ResetExe,
    Busy => GVL_AXIS1.stBC_Reset.Busy,
    Error => GVL_AXIS1.stBC_Reset.Error,
    ErrorID => GVL_AXIS1.stBC_Reset.ErrorID); // MC_Reset
GVL_AXIS1.stBC_Reset.Done := GVL_AXIS1.fbBC_Reset.Done;

// NETWORK 3

// NETWORK 4
GVL_AXIS1.fbBC_Power(
    Axis := GVL_AXIS1.BCAxis,
    Enable := GVL_AXIS1.bBC_PowerEnCmd,
    Enable_Positive := GVL_AXIS1.bBC_PowerEnPositive,
    Enable_Negative := GVL_AXIS1.bBC_PowerEnNegative,
    Override := GVL_AXIS1.lrBC_PowerOverride,
    Busy => GVL_AXIS1.stBC_Power.Busy,
    Active => GVL_AXIS1.stBC_Power.Active,
    Error => GVL_AXIS1.stBC_Power.Error,
    ErrorID => GVL_AXIS1.stBC_Power.ErrorID); // MC_Power
GVL_AXIS1.stBC_Power.Status := GVL_AXIS1.fbBC_Power.Status;

// NETWORK 5
GVL_AXIS1.fbBC_MoveVelocity(
    Axis := GVL_AXIS1.BCAxis,
    Execute := GVL_AXIS1.stBC_VelCmd.bExe,
    Velocity := GVL_AXIS1.stBC_VelCmd.lrVelocity,
    Acceleration := GVL_AXIS1.stBC_VelCmd.lrAcceleration,
    Deceleration := GVL_AXIS1.stBC_VelCmd.lrDeceleration,
    Jerk := GVL_AXIS1.stBC_VelCmd.lrJerk,
    Direction := GVL_AXIS1.stBC_VelCmd.EnuDirection,
    BufferMode := GVL_AXIS1.stBC_VelCmd.EnuBufferMode,
    Options := GVL_AXIS1.stBC_VelCmd.EnuOptions,
    Busy => GVL_AXIS1.stBC_MoveVelocity.Busy,
    Active => GVL_AXIS1.stBC_MoveVelocity.Active,
    CommandAborted => GVL_AXIS1.stBC_MoveVelocity.CmdAborted,
    Error => GVL_AXIS1.stBC_MoveVelocity.Error,
    ErrorID => GVL_AXIS1.stBC_MoveVelocity.ErrorID); // MC_MoveVelocity
GVL_AXIS1.stBC_MoveVelocity.InVelocity := GVL_AXIS1.fbBC_MoveVelocity.InVelocity;

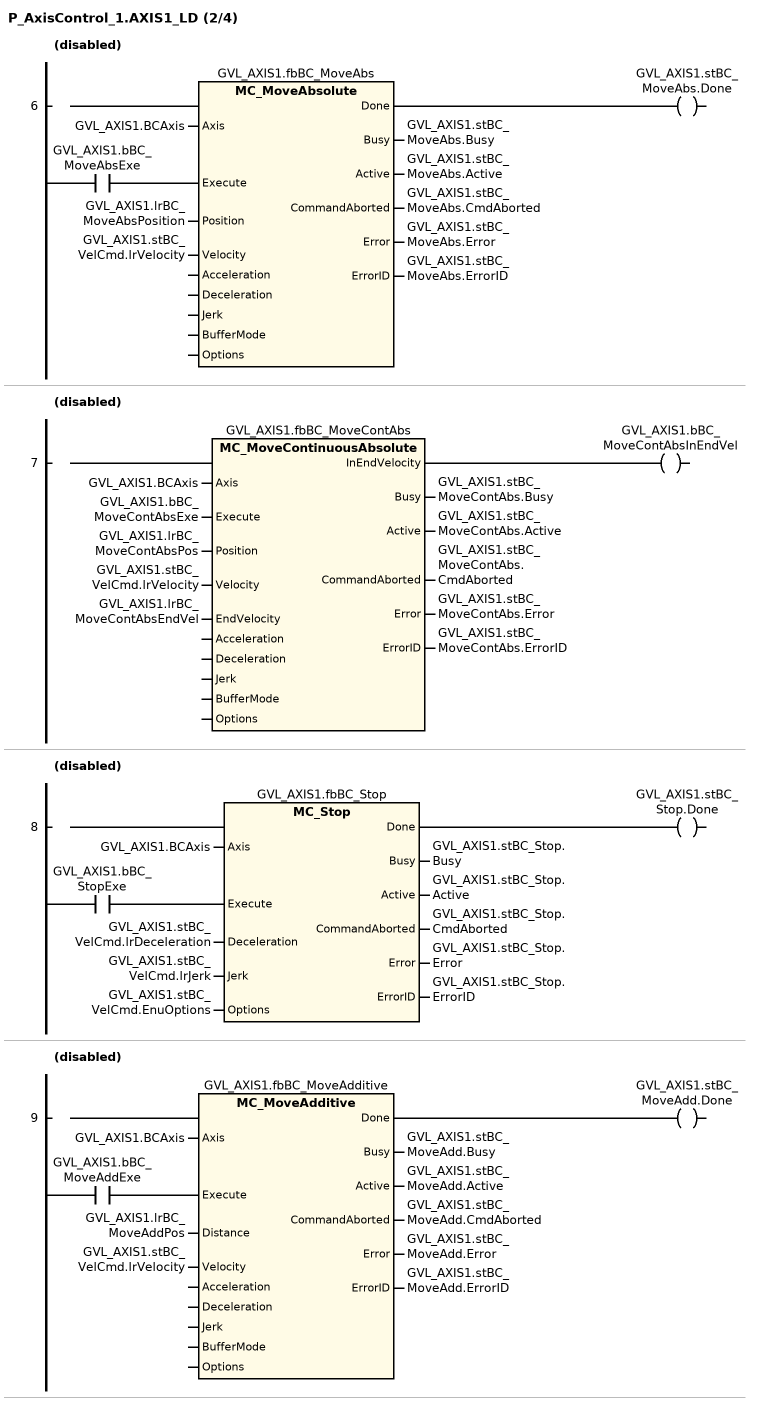
// NETWORK 6 (disabled)
// GVL_AXIS1.fbBC_MoveAbs(
//     Axis := GVL_AXIS1.BCAxis,
//     Execute := GVL_AXIS1.bBC_MoveAbsExe,
//     Position := GVL_AXIS1.lrBC_MoveAbsPosition,
//     Velocity := GVL_AXIS1.stBC_VelCmd.lrVelocity,
//     Busy => GVL_AXIS1.stBC_MoveAbs.Busy,
//     Active => GVL_AXIS1.stBC_MoveAbs.Active,
//     CommandAborted => GVL_AXIS1.stBC_MoveAbs.CmdAborted,
//     Error => GVL_AXIS1.stBC_MoveAbs.Error,
//     ErrorID => GVL_AXIS1.stBC_MoveAbs.ErrorID); // MC_MoveAbsolute
// GVL_AXIS1.stBC_MoveAbs.Done := GVL_AXIS1.fbBC_MoveAbs.Done;

// NETWORK 7 (disabled)
// GVL_AXIS1.fbBC_MoveContAbs(
//     Axis := GVL_AXIS1.BCAxis,
//     Execute := GVL_AXIS1.bBC_MoveContAbsExe,
//     Position := GVL_AXIS1.lrBC_MoveContAbsPos,
//     Velocity := GVL_AXIS1.stBC_VelCmd.lrVelocity,
//     EndVelocity := GVL_AXIS1.lrBC_MoveContAbsEndVel,
//     Busy => GVL_AXIS1.stBC_MoveContAbs.Busy,
//     Active => GVL_AXIS1.stBC_MoveContAbs.Active,
//     CommandAborted => GVL_AXIS1.stBC_MoveContAbs.CmdAborted,
//     Error => GVL_AXIS1.stBC_MoveContAbs.Error,
//     ErrorID => GVL_AXIS1.stBC_MoveContAbs.ErrorID); // MC_MoveContinuousAbsolute
// GVL_AXIS1.bBC_MoveContAbsInEndVel := GVL_AXIS1.fbBC_MoveContAbs.InEndVelocity;

// NETWORK 8 (disabled)
// GVL_AXIS1.fbBC_Stop(
//     Axis := GVL_AXIS1.BCAxis,
//     Execute := GVL_AXIS1.bBC_StopExe,
//     Deceleration := GVL_AXIS1.stBC_VelCmd.lrDeceleration,
//     Jerk := GVL_AXIS1.stBC_VelCmd.lrJerk,
//     Options := GVL_AXIS1.stBC_VelCmd.EnuOptions,
//     Busy => GVL_AXIS1.stBC_Stop.Busy,
//     Active => GVL_AXIS1.stBC_Stop.Active,
//     CommandAborted => GVL_AXIS1.stBC_Stop.CmdAborted,
//     Error => GVL_AXIS1.stBC_Stop.Error,
//     ErrorID => GVL_AXIS1.stBC_Stop.ErrorID); // MC_Stop
// GVL_AXIS1.stBC_Stop.Done := GVL_AXIS1.fbBC_Stop.Done;

// NETWORK 9 (disabled)
// GVL_AXIS1.fbBC_MoveAdditive(
//     Axis := GVL_AXIS1.BCAxis,
//     Execute := GVL_AXIS1.bBC_MoveAddExe,
//     Distance := GVL_AXIS1.lrBC_MoveAddPos,
//     Velocity := GVL_AXIS1.stBC_VelCmd.lrVelocity,
//     Busy => GVL_AXIS1.stBC_MoveAdd.Busy,
//     Active => GVL_AXIS1.stBC_MoveAdd.Active,
//     CommandAborted => GVL_AXIS1.stBC_MoveAdd.CmdAborted,
//     Error => GVL_AXIS1.stBC_MoveAdd.Error,
//     ErrorID => GVL_AXIS1.stBC_MoveAdd.ErrorID); // MC_MoveAdditive
// GVL_AXIS1.stBC_MoveAdd.Done := GVL_AXIS1.fbBC_MoveAdditive.Done;

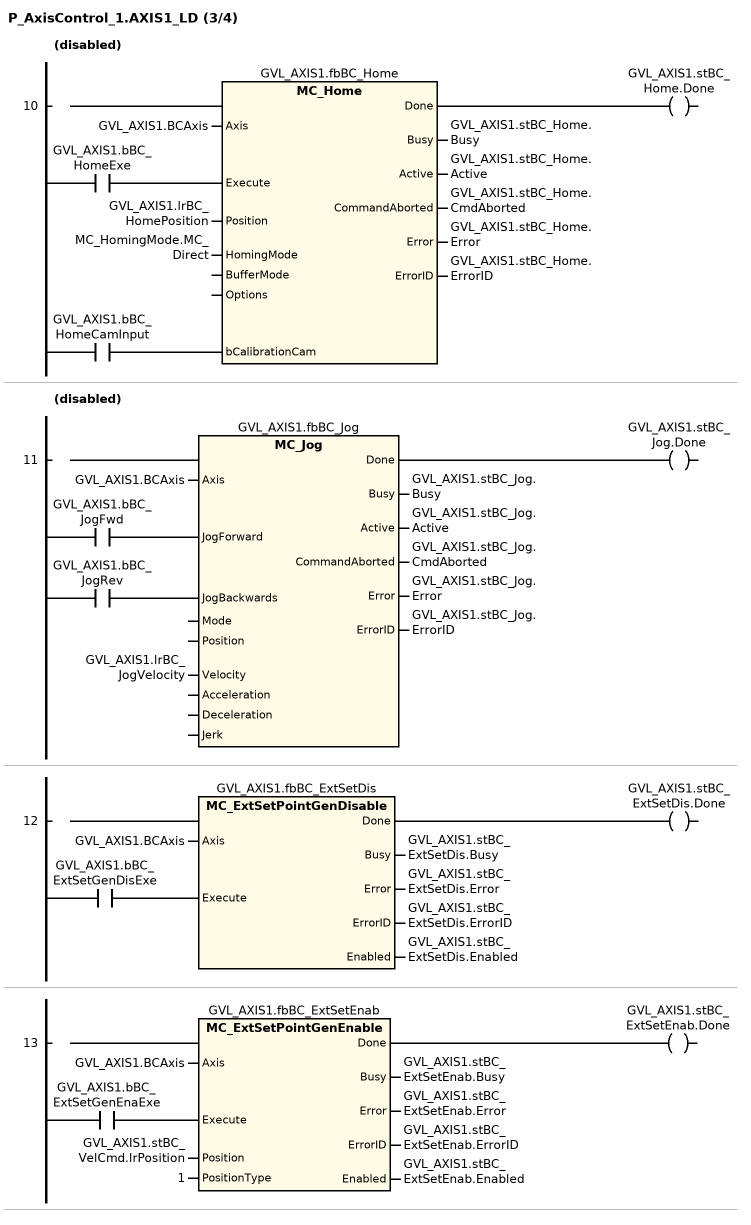
// NETWORK 10 (disabled)
// GVL_AXIS1.fbBC_Home(
//     Axis := GVL_AXIS1.BCAxis,
//     Execute := GVL_AXIS1.bBC_HomeExe,
//     Position := GVL_AXIS1.lrBC_HomePosition,
//     HomingMode := MC_HomingMode.MC_Direct,
//     bCalibrationCam := GVL_AXIS1.bBC_HomeCamInput,
//     Busy => GVL_AXIS1.stBC_Home.Busy,
//     Active => GVL_AXIS1.stBC_Home.Active,
//     CommandAborted => GVL_AXIS1.stBC_Home.CmdAborted,
//     Error => GVL_AXIS1.stBC_Home.Error,
//     ErrorID => GVL_AXIS1.stBC_Home.ErrorID); // MC_Home
// GVL_AXIS1.stBC_Home.Done := GVL_AXIS1.fbBC_Home.Done;

// NETWORK 11 (disabled)
// GVL_AXIS1.fbBC_Jog(
//     Axis := GVL_AXIS1.BCAxis,
//     JogForward := GVL_AXIS1.bBC_JogFwd,
//     JogBackwards := GVL_AXIS1.bBC_JogRev,
//     Velocity := GVL_AXIS1.lrBC_JogVelocity,
//     Busy => GVL_AXIS1.stBC_Jog.Busy,
//     Active => GVL_AXIS1.stBC_Jog.Active,
//     CommandAborted => GVL_AXIS1.stBC_Jog.CmdAborted,
//     Error => GVL_AXIS1.stBC_Jog.Error,
//     ErrorID => GVL_AXIS1.stBC_Jog.ErrorID); // MC_Jog
// GVL_AXIS1.stBC_Jog.Done := GVL_AXIS1.fbBC_Jog.Done;

// NETWORK 12
GVL_AXIS1.fbBC_ExtSetDis(
    Axis := GVL_AXIS1.BCAxis,
    Execute := GVL_AXIS1.bBC_ExtSetGenDisExe,
    Busy => GVL_AXIS1.stBC_ExtSetDis.Busy,
    Error => GVL_AXIS1.stBC_ExtSetDis.Error,
    ErrorID => GVL_AXIS1.stBC_ExtSetDis.ErrorID,
    Enabled => GVL_AXIS1.stBC_ExtSetDis.Enabled); // MC_ExtSetPointGenDisable
GVL_AXIS1.stBC_ExtSetDis.Done := GVL_AXIS1.fbBC_ExtSetDis.Done;

// NETWORK 13
GVL_AXIS1.fbBC_ExtSetEnab(
    Axis := GVL_AXIS1.BCAxis,
    Execute := GVL_AXIS1.bBC_ExtSetGenEnaExe,
    Position := GVL_AXIS1.stBC_VelCmd.lrPosition,
    PositionType := 1,
    Busy => GVL_AXIS1.stBC_ExtSetEnab.Busy,
    Error => GVL_AXIS1.stBC_ExtSetEnab.Error,
    ErrorID => GVL_AXIS1.stBC_ExtSetEnab.ErrorID,
    Enabled => GVL_AXIS1.stBC_ExtSetEnab.Enabled); // MC_ExtSetPointGenEnable
GVL_AXIS1.stBC_ExtSetEnab.Done := GVL_AXIS1.fbBC_ExtSetEnab.Done;

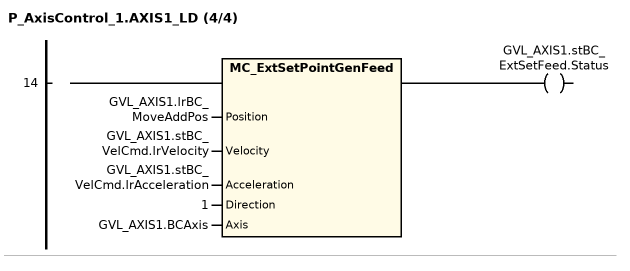
// NETWORK 14
GVL_AXIS1.stBC_ExtSetFeed.Status := MC_ExtSetPointGenFeed(Position := GVL_AXIS1.lrBC_MoveAddPos, Velocity := GVL_AXIS1.stBC_VelCmd.lrVelocity, Acceleration := GVL_AXIS1.stBC_VelCmd.lrAcceleration, Direction := 1, Axis := GVL_AXIS1.BCAxis);
END_METHOD

METHOD AXIS2_LD : BOOL
VAR_INPUT
END_VAR
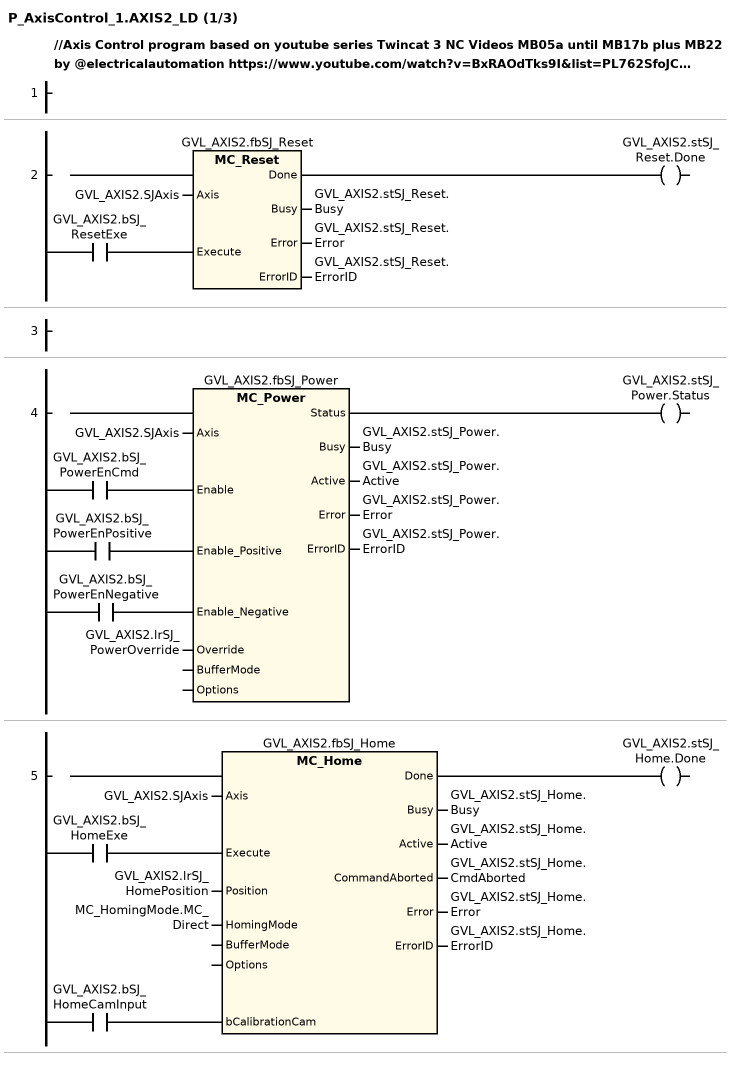
// NETWORK 1: //Axis Control program based on youtube series Twincat 3 NC Videos MB05a until MB17b plus MB22 by @electricalautomation https://www.youtube.com/watch?v=BxRAOdTks9I&list=PL762SfoJC-e8NbAUQ-H7a_TOdqrlBPCw4&index=25

// NETWORK 2
GVL_AXIS2.fbSJ_Reset(
    Axis := GVL_AXIS2.SJAxis,
    Execute := GVL_AXIS2.bSJ_ResetExe,
    Busy => GVL_AXIS2.stSJ_Reset.Busy,
    Error => GVL_AXIS2.stSJ_Reset.Error,
    ErrorID => GVL_AXIS2.stSJ_Reset.ErrorID); // MC_Reset
GVL_AXIS2.stSJ_Reset.Done := GVL_AXIS2.fbSJ_Reset.Done;

// NETWORK 3

// NETWORK 4
GVL_AXIS2.fbSJ_Power(
    Axis := GVL_AXIS2.SJAxis,
    Enable := GVL_AXIS2.bSJ_PowerEnCmd,
    Enable_Positive := GVL_AXIS2.bSJ_PowerEnPositive,
    Enable_Negative := GVL_AXIS2.bSJ_PowerEnNegative,
    Override := GVL_AXIS2.lrSJ_PowerOverride,
    Busy => GVL_AXIS2.stSJ_Power.Busy,
    Active => GVL_AXIS2.stSJ_Power.Active,
    Error => GVL_AXIS2.stSJ_Power.Error,
    ErrorID => GVL_AXIS2.stSJ_Power.ErrorID); // MC_Power
GVL_AXIS2.stSJ_Power.Status := GVL_AXIS2.fbSJ_Power.Status;

// NETWORK 5
GVL_AXIS2.fbSJ_Home(
    Axis := GVL_AXIS2.SJAxis,
    Execute := GVL_AXIS2.bSJ_HomeExe,
    Position := GVL_AXIS2.lrSJ_HomePosition,
    HomingMode := MC_HomingMode.MC_Direct,
    bCalibrationCam := GVL_AXIS2.bSJ_HomeCamInput,
    Busy => GVL_AXIS2.stSJ_Home.Busy,
    Active => GVL_AXIS2.stSJ_Home.Active,
    CommandAborted => GVL_AXIS2.stSJ_Home.CmdAborted,
    Error => GVL_AXIS2.stSJ_Home.Error,
    ErrorID => GVL_AXIS2.stSJ_Home.ErrorID); // MC_Home
GVL_AXIS2.stSJ_Home.Done := GVL_AXIS2.fbSJ_Home.Done;

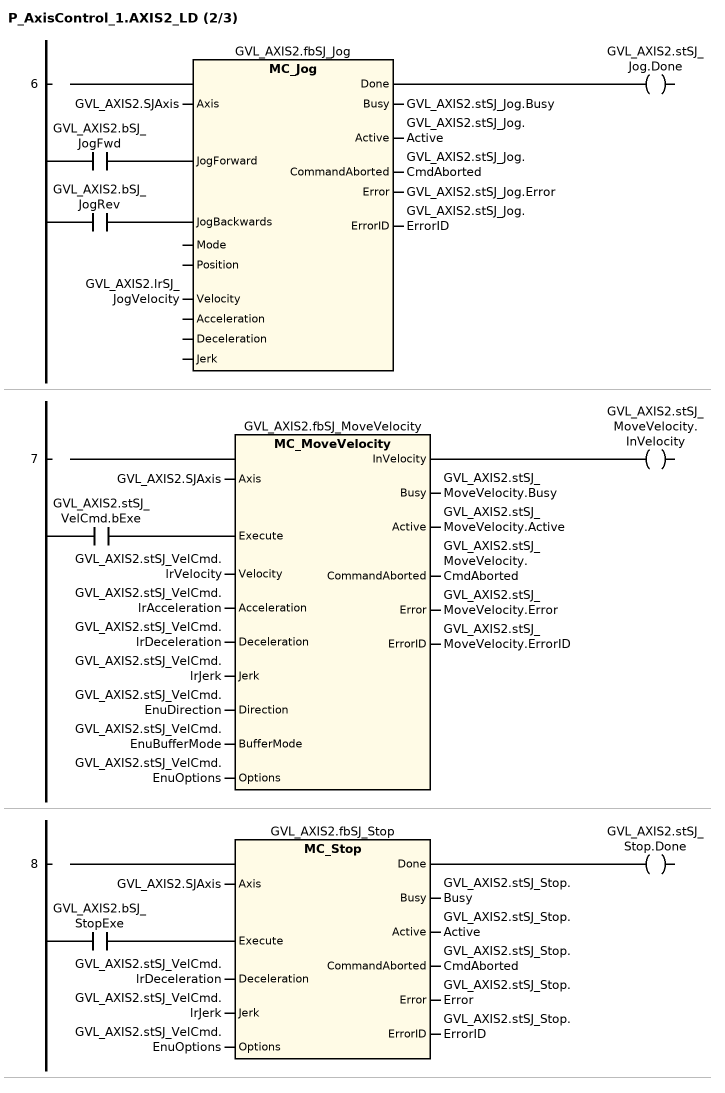
// NETWORK 6
GVL_AXIS2.fbSJ_Jog(
    Axis := GVL_AXIS2.SJAxis,
    JogForward := GVL_AXIS2.bSJ_JogFwd,
    JogBackwards := GVL_AXIS2.bSJ_JogRev,
    Velocity := GVL_AXIS2.lrSJ_JogVelocity,
    Busy => GVL_AXIS2.stSJ_Jog.Busy,
    Active => GVL_AXIS2.stSJ_Jog.Active,
    CommandAborted => GVL_AXIS2.stSJ_Jog.CmdAborted,
    Error => GVL_AXIS2.stSJ_Jog.Error,
    ErrorID => GVL_AXIS2.stSJ_Jog.ErrorID); // MC_Jog
GVL_AXIS2.stSJ_Jog.Done := GVL_AXIS2.fbSJ_Jog.Done;

// NETWORK 7
GVL_AXIS2.fbSJ_MoveVelocity(
    Axis := GVL_AXIS2.SJAxis,
    Execute := GVL_AXIS2.stSJ_VelCmd.bExe,
    Velocity := GVL_AXIS2.stSJ_VelCmd.lrVelocity,
    Acceleration := GVL_AXIS2.stSJ_VelCmd.lrAcceleration,
    Deceleration := GVL_AXIS2.stSJ_VelCmd.lrDeceleration,
    Jerk := GVL_AXIS2.stSJ_VelCmd.lrJerk,
    Direction := GVL_AXIS2.stSJ_VelCmd.EnuDirection,
    BufferMode := GVL_AXIS2.stSJ_VelCmd.EnuBufferMode,
    Options := GVL_AXIS2.stSJ_VelCmd.EnuOptions,
    Busy => GVL_AXIS2.stSJ_MoveVelocity.Busy,
    Active => GVL_AXIS2.stSJ_MoveVelocity.Active,
    CommandAborted => GVL_AXIS2.stSJ_MoveVelocity.CmdAborted,
    Error => GVL_AXIS2.stSJ_MoveVelocity.Error,
    ErrorID => GVL_AXIS2.stSJ_MoveVelocity.ErrorID); // MC_MoveVelocity
GVL_AXIS2.stSJ_MoveVelocity.InVelocity := GVL_AXIS2.fbSJ_MoveVelocity.InVelocity;

// NETWORK 8
GVL_AXIS2.fbSJ_Stop(
    Axis := GVL_AXIS2.SJAxis,
    Execute := GVL_AXIS2.bSJ_StopExe,
    Deceleration := GVL_AXIS2.stSJ_VelCmd.lrDeceleration,
    Jerk := GVL_AXIS2.stSJ_VelCmd.lrJerk,
    Options := GVL_AXIS2.stSJ_VelCmd.EnuOptions,
    Busy => GVL_AXIS2.stSJ_Stop.Busy,
    Active => GVL_AXIS2.stSJ_Stop.Active,
    CommandAborted => GVL_AXIS2.stSJ_Stop.CmdAborted,
    Error => GVL_AXIS2.stSJ_Stop.Error,
    ErrorID => GVL_AXIS2.stSJ_Stop.ErrorID); // MC_Stop
GVL_AXIS2.stSJ_Stop.Done := GVL_AXIS2.fbSJ_Stop.Done;

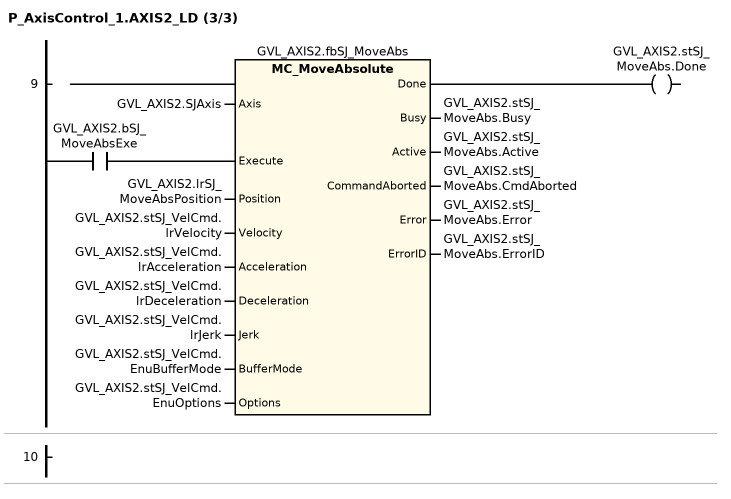
// NETWORK 9
GVL_AXIS2.fbSJ_MoveAbs(
    Axis := GVL_AXIS2.SJAxis,
    Execute := GVL_AXIS2.bSJ_MoveAbsExe,
    Position := GVL_AXIS2.lrSJ_MoveAbsPosition,
    Velocity := GVL_AXIS2.stSJ_VelCmd.lrVelocity,
    Acceleration := GVL_AXIS2.stSJ_VelCmd.lrAcceleration,
    Deceleration := GVL_AXIS2.stSJ_VelCmd.lrDeceleration,
    Jerk := GVL_AXIS2.stSJ_VelCmd.lrJerk,
    BufferMode := GVL_AXIS2.stSJ_VelCmd.EnuBufferMode,
    Options := GVL_AXIS2.stSJ_VelCmd.EnuOptions,
    Busy => GVL_AXIS2.stSJ_MoveAbs.Busy,
    Active => GVL_AXIS2.stSJ_MoveAbs.Active,
    CommandAborted => GVL_AXIS2.stSJ_MoveAbs.CmdAborted,
    Error => GVL_AXIS2.stSJ_MoveAbs.Error,
    ErrorID => GVL_AXIS2.stSJ_MoveAbs.ErrorID); // MC_MoveAbsolute
GVL_AXIS2.stSJ_MoveAbs.Done := GVL_AXIS2.fbSJ_MoveAbs.Done;

// NETWORK 10
END_METHOD

METHOD AXIS3_LD : BOOL
VAR_INPUT
END_VAR
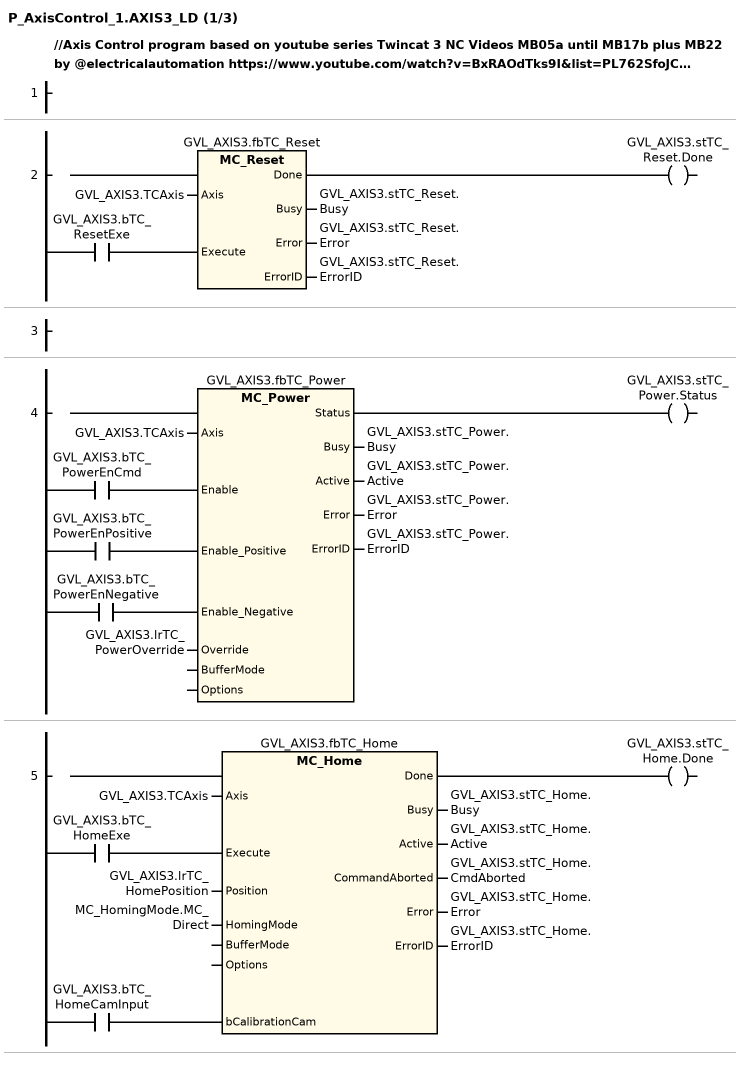
// NETWORK 1: //Axis Control program based on youtube series Twincat 3 NC Videos MB05a until MB17b plus MB22 by @electricalautomation https://www.youtube.com/watch?v=BxRAOdTks9I&list=PL762SfoJC-e8NbAUQ-H7a_TOdqrlBPCw4&index=25

// NETWORK 2
GVL_AXIS3.fbTC_Reset(
    Axis := GVL_AXIS3.TCAxis,
    Execute := GVL_AXIS3.bTC_ResetExe,
    Busy => GVL_AXIS3.stTC_Reset.Busy,
    Error => GVL_AXIS3.stTC_Reset.Error,
    ErrorID => GVL_AXIS3.stTC_Reset.ErrorID); // MC_Reset
GVL_AXIS3.stTC_Reset.Done := GVL_AXIS3.fbTC_Reset.Done;

// NETWORK 3

// NETWORK 4
GVL_AXIS3.fbTC_Power(
    Axis := GVL_AXIS3.TCAxis,
    Enable := GVL_AXIS3.bTC_PowerEnCmd,
    Enable_Positive := GVL_AXIS3.bTC_PowerEnPositive,
    Enable_Negative := GVL_AXIS3.bTC_PowerEnNegative,
    Override := GVL_AXIS3.lrTC_PowerOverride,
    Busy => GVL_AXIS3.stTC_Power.Busy,
    Active => GVL_AXIS3.stTC_Power.Active,
    Error => GVL_AXIS3.stTC_Power.Error,
    ErrorID => GVL_AXIS3.stTC_Power.ErrorID); // MC_Power
GVL_AXIS3.stTC_Power.Status := GVL_AXIS3.fbTC_Power.Status;

// NETWORK 5
GVL_AXIS3.fbTC_Home(
    Axis := GVL_AXIS3.TCAxis,
    Execute := GVL_AXIS3.bTC_HomeExe,
    Position := GVL_AXIS3.lrTC_HomePosition,
    HomingMode := MC_HomingMode.MC_Direct,
    bCalibrationCam := GVL_AXIS3.bTC_HomeCamInput,
    Busy => GVL_AXIS3.stTC_Home.Busy,
    Active => GVL_AXIS3.stTC_Home.Active,
    CommandAborted => GVL_AXIS3.stTC_Home.CmdAborted,
    Error => GVL_AXIS3.stTC_Home.Error,
    ErrorID => GVL_AXIS3.stTC_Home.ErrorID); // MC_Home
GVL_AXIS3.stTC_Home.Done := GVL_AXIS3.fbTC_Home.Done;

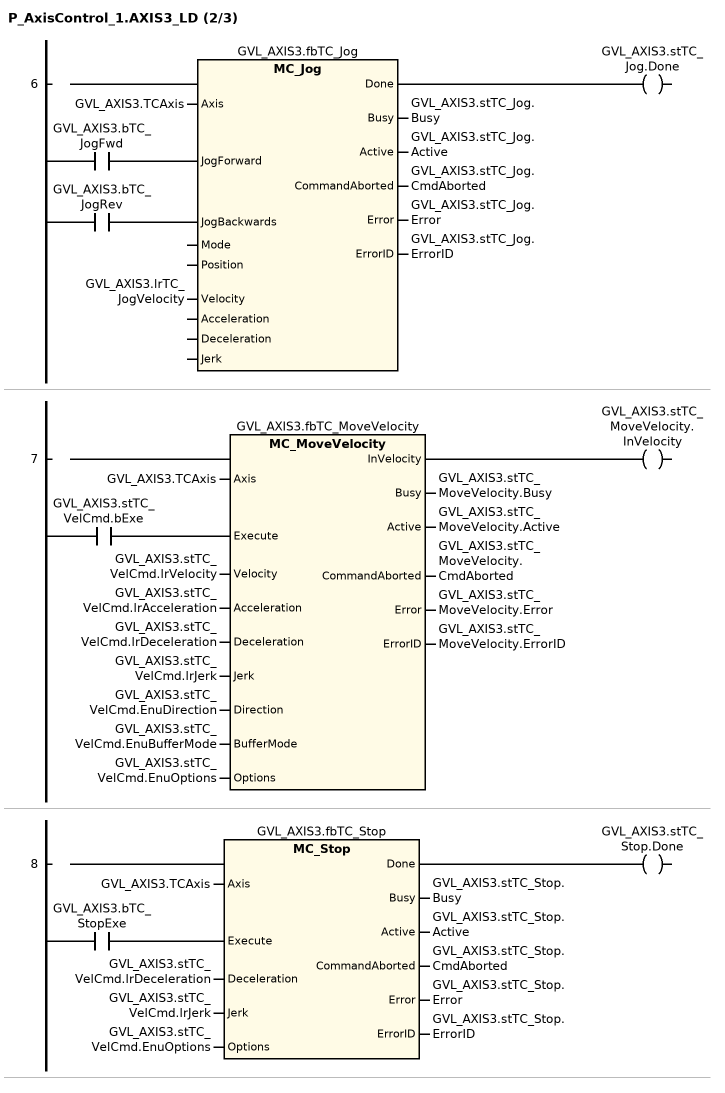
// NETWORK 6
GVL_AXIS3.fbTC_Jog(
    Axis := GVL_AXIS3.TCAxis,
    JogForward := GVL_AXIS3.bTC_JogFwd,
    JogBackwards := GVL_AXIS3.bTC_JogRev,
    Velocity := GVL_AXIS3.lrTC_JogVelocity,
    Busy => GVL_AXIS3.stTC_Jog.Busy,
    Active => GVL_AXIS3.stTC_Jog.Active,
    CommandAborted => GVL_AXIS3.stTC_Jog.CmdAborted,
    Error => GVL_AXIS3.stTC_Jog.Error,
    ErrorID => GVL_AXIS3.stTC_Jog.ErrorID); // MC_Jog
GVL_AXIS3.stTC_Jog.Done := GVL_AXIS3.fbTC_Jog.Done;

// NETWORK 7
GVL_AXIS3.fbTC_MoveVelocity(
    Axis := GVL_AXIS3.TCAxis,
    Execute := GVL_AXIS3.stTC_VelCmd.bExe,
    Velocity := GVL_AXIS3.stTC_VelCmd.lrVelocity,
    Acceleration := GVL_AXIS3.stTC_VelCmd.lrAcceleration,
    Deceleration := GVL_AXIS3.stTC_VelCmd.lrDeceleration,
    Jerk := GVL_AXIS3.stTC_VelCmd.lrJerk,
    Direction := GVL_AXIS3.stTC_VelCmd.EnuDirection,
    BufferMode := GVL_AXIS3.stTC_VelCmd.EnuBufferMode,
    Options := GVL_AXIS3.stTC_VelCmd.EnuOptions,
    Busy => GVL_AXIS3.stTC_MoveVelocity.Busy,
    Active => GVL_AXIS3.stTC_MoveVelocity.Active,
    CommandAborted => GVL_AXIS3.stTC_MoveVelocity.CmdAborted,
    Error => GVL_AXIS3.stTC_MoveVelocity.Error,
    ErrorID => GVL_AXIS3.stTC_MoveVelocity.ErrorID); // MC_MoveVelocity
GVL_AXIS3.stTC_MoveVelocity.InVelocity := GVL_AXIS3.fbTC_MoveVelocity.InVelocity;

// NETWORK 8
GVL_AXIS3.fbTC_Stop(
    Axis := GVL_AXIS3.TCAxis,
    Execute := GVL_AXIS3.bTC_StopExe,
    Deceleration := GVL_AXIS3.stTC_VelCmd.lrDeceleration,
    Jerk := GVL_AXIS3.stTC_VelCmd.lrJerk,
    Options := GVL_AXIS3.stTC_VelCmd.EnuOptions,
    Busy => GVL_AXIS3.stTC_Stop.Busy,
    Active => GVL_AXIS3.stTC_Stop.Active,
    CommandAborted => GVL_AXIS3.stTC_Stop.CmdAborted,
    Error => GVL_AXIS3.stTC_Stop.Error,
    ErrorID => GVL_AXIS3.stTC_Stop.ErrorID); // MC_Stop
GVL_AXIS3.stTC_Stop.Done := GVL_AXIS3.fbTC_Stop.Done;

